// TwinCAT 3 PLC project FsCommon
// Title: FsCommon
// Company: FisoThemes
// Author: Goodwill Mzumala
// ProjectVersion: 0.7.0
// Description: A library that contains common utilites and definitiions to streamline and standardise the development of PLC applications.
// ProgramVersion: 3.1.4023.0
// libraries:
//   SysTarget, * (System)
//   Tc2_Math, * (Beckhoff Automation GmbH)
//   Tc2_Standard, * (Beckhoff Automation GmbH)
//   Tc2_System, * (Beckhoff Automation GmbH)
//   Tc3_Module, * (Beckhoff Automation GmbH)
// project tree:
//   DUTs/ E_Accessor.TcTLEO, E_Comparison.TcTLEO, E_AddressMemoryArea.TcTLEO, E_OperatingSystem.TcTLEO, E_ProcessorArchitecture.TcTLEO, ST_ArrayIterator.TcDUT, T_ArrayIterator.TcDUT, T_Path.TcDUT, T_TypeID.TcDUT, T_WPath.TcDUT, U_Primitive.TcDUT, T_Char.TcDUT, T_MaxWString.TcDUT, T_WChar.TcDUT, T_Generic.TcDUT, T_TaskNameString.TcDUT, T_TypeClass.TcDUT, T_PlcAppSysInfo.TcDUT, T_Position.TcDUT, T_QueryInterface.TcDUT, T_Size.TcDUT, T_VarInfo.TcDUT, U_Pointer.TcDUT
//   DUTs/Primitives/ F32.TcDUT, F64.TcDUT, I16.TcDUT, I32.TcDUT, I64.TcDUT, I8.TcDUT, U16.TcDUT, U32.TcDUT, U64.TcDUT, U8.TcDUT
//   GVLs/ GVL_TypeValueLimits.TcGVL
//   ITFs/ I_ChangeDetector.TcIO, I_PlcTaskInformation.TcIO, I_Destructable.TcIO, I_Runnable.TcIO
//   PARAMs/ PARAM_Constants.TcGVL
//   / PlcTask.TcTTO
//   POUs/Bounds/ F_GetBoolArrayUpperBound.TcPOU, F_GetByteArrayUpperBound.TcPOU, F_GetDateAndTimeArrayUpperBound.TcPOU, F_GetDateArrayUpperBound.TcPOU, F_GetDIntArrayUpperBound.TcPOU, F_GetDWordArrayUpperBound.TcPOU, F_GetIntArrayUpperBound.TcPOU, F_GetInterfaceArrayLowerBound.TcPOU, F_GetInterfaceArrayUpperBound.TcPOU, F_GetLIntArrayUpperBound.TcPOU, F_GetLRealArrayUpperBound.TcPOU, F_GetLTimeArrayUpperBound.TcPOU, F_GetLWordArrayUpperBound.TcPOU, F_GetMaxStringArrayLowerBound.TcPOU, F_GetMaxStringArrayUpperBound.TcPOU, F_GetMaxWStringArrayLowerBound.TcPOU, F_GetMaxWStringArrayUpperBound.TcPOU, F_GetPointerArrayUpperBound.TcPOU, F_GetRealArrayUpperBound.TcPOU, F_GetRunnableArrayLowerBound.TcPOU, F_GetRunnableArrayUpperBound.TcPOU, F_GetSIntArrayUpperBound.TcPOU, F_GetStringArrayUpperBound.TcPOU, F_GetTimeArrayUpperBound.TcPOU, F_GetTimeOfDayArrayUpperBound.TcPOU, F_GetUDIntArrayUpperBound.TcPOU, F_GetUIntArrayUpperBound.TcPOU, F_GetULIntArrayUpperBound.TcPOU, F_GetUSIntArrayUpperBound.TcPOU, F_GetUXIntArrayUpperBound.TcPOU, F_GetWordArrayUpperBound.TcPOU, F_GetWStringArrayLowerBound.TcPOU, F_GetStringArrayLowerBound.TcPOU, F_GetPointerArrayLowerBound.TcPOU, F_GetTimeOfDayArrayLowerBound.TcPOU, F_GetDateAndTimeArrayLowerBound.TcPOU, F_GetDateArrayLowerBound.TcPOU, F_GetTimeArrayLowerBound.TcPOU, F_GetRealArrayLowerBound.TcPOU, F_GetLRealArrayLowerBound.TcPOU, F_GetLTimeArrayLowerBound.TcPOU, F_GetUDIntArrayLowerBound.TcPOU, F_GetULIntArrayLowerBound.TcPOU, F_GetUXIntArrayLowerBound.TcPOU, F_GetUSIntArrayLowerBound.TcPOU, F_GetDIntArrayLowerBound.TcPOU, F_GetLIntArrayLowerBound.TcPOU, F_GetUIntArrayLowerBound.TcPOU, F_GetWStringArrayUpperBound.TcPOU, F_GetXIntArrayLowerBound.TcPOU, F_GetSIntArrayLowerBound.TcPOU, F_GetByteArrayLowerBound.TcPOU, F_GetBoolArrayLowerBound.TcPOU, F_GetLWordArrayLowerBound.TcPOU, F_GetIntArrayLowerBound.TcPOU, F_GetXIntArrayUpperBound.TcPOU, F_GetXWordArrayLowerBound.TcPOU, F_GetWordArrayLowerBound.TcPOU, F_GetDWordArrayLowerBound.TcPOU, F_GetXWordArrayUpperBound.TcPOU
//   POUs/Conversions/ F_DintToSize.TcPOU, F_IntToSize.TcPOU, F_PositionToSize.TcPOU (not stored), F_SizeToDint.TcPOU (not stored), F_SizeToInt.TcPOU (not stored), F_SizeToPosition.TcPOU, F_ULintToPosition.TcPOU
//   POUs/ FB_PlcTaskInformation.TcPOU, FB_RandomNumberGenerator.TcPOU, FB_ValueChangeDetector.TcPOU, FB_PlcTaskCycleChangeDetector.TcPOU, F_AllAreFalse.TcPOU, F_AllocateMemory.TcPOU, F_AnyAreTrue.TcPOU, F_AnyAreFalse.TcPOU, F_AreSameTypeFromInterfaces.TcPOU, F_ExtractPointerFromInterface.TcPOU, F_ExtractVariableNameFromPath.TcPOU, F_GetAddressMemoryArea.TcPOU, F_GetCpuCycleCounter.TcPOU, F_GetCurrentTaskCycleTime.TcPOU, F_GetCurrentPlcTaskInformation.TcPOU, F_GetCurrentTaskIndex.TcPOU, F_GetInf.TcPOU, F_GetMemorySegment.TcPOU, F_GetNaN.TcPOU, F_GetAddressFromInterface.TcPOU, F_DeallocateMemory.TcPOU, F_GetNumberOfPlcTasks.TcPOU, F_GetTypeID.TcPOU, F_GetTypeIDFromGeneric.TcPOU, F_GetVariablePathByAddress.TcPOU, F_GetVariablePath.TcPOU, F_Hash.TcPOU, F_AllAreTrue.TcPOU, F_IsPointerToFunctionBlock.TcPOU, F_IsPointerToInterface.TcPOU, F_IsReadablePointer.TcPOU, F_Lerp.TcPOU, F_ResetOnTrue.TcPOU, F_RunAllRunnables.TcPOU, F_SearchMemory.TcPOU, F_SetDecimalPlaces.TcPOU, F_SetOnFalse.TcPOU, F_SwapMemory.TcPOU, FB_TcComIecApplicationInfo.TcPOU, F_GetTypeNameByAddress.TcPOU, F_GetTypeName.TcPOU, F_GetTypeNameByPath.TcPOU, F_TcComIecApplicationInfo.TcPOU, F_RoundToDecimalPlaces.TcPOU, F_TruncateNumber.TcPOU, F_TryDerefPointer.TcPOU, P_GetSystemInformation.TcPOU, PLAYGROUND.TcPOU
//   Project Information/ F_GetCompany.TcPOU, F_GetTitle.TcPOU, F_GetVersion.TcPOU
//   Version/ Global_Version.TcGVL
// real-time tasks:
//   TASK PlcTask: cycle T#10ms, priority 20, ADS port 350
//   TASK PlcTestTask: cycle T#10ms, priority 21, ADS port 351

CONFIGURATION FsCommon
    RESOURCE PLC ON TwinCAT3
        TASK PlcTask(INTERVAL := T#10ms, PRIORITY := 20);
        PROGRAM PLAYGROUND WITH PlcTask : PLAYGROUND;
    END_RESOURCE
END_CONFIGURATION

// ---- DUTs/E_Accessor.TcTLEO
// An enum that can be used to represent getters and setters.
{attribute 'qualified_only'}
{attribute 'to_string'}
TYPE E_Accessor :
(
	_ := 0, // Unknown/Invalid
	Get,
	Set
)BYTE;
END_TYPE

// ---- DUTs/E_Comparison.TcTLEO
// Comparison enum.
{attribute 'qualified_only'}
{attribute 'to_string'}
TYPE E_Comparison :
(
	_ := 0, // Unknown/Invalid
	Less,
	Equal,
	Greater
)BYTE;
END_TYPE

// ---- DUTs/E_AddressMemoryArea.TcTLEO
// An enum to specify the memory area type of an address.
{attribute 'qualified_only'}
{attribute 'to_string'}
TYPE E_AddressMemoryArea :
(
	_ 		:= 0, 	// Unknown/Invalid.
	Static	:= 1, 	// Static memory.
	Dynamic	:= 2, 	// Dynamic memory.
	CNC		:= 3	// CNC static memory.
)BYTE;
END_TYPE

// ---- DUTs/E_OperatingSystem.TcTLEO
// Operating system used by the machine.
{attribute 'qualified_only'}
{attribute 'to_string'}
TYPE E_OperatingSystem :
(
	_ 			:= 0, 		// Invalid/Unknown/Ininitialised
	Windows,				// Windows OS
	Linux		:= 5,		// Linux
	VxWorks,				// VxWorks RTOS
	QNX,					// Blackberry QNX Embedded OS
	uCOS					// Micro-Controller Operating Systems by Jean J. Labrosse (1991)
) BYTE;
END_TYPE

// ---- DUTs/E_ProcessorArchitecture.TcTLEO
// Processor used by the machine.
{attribute 'qualified_only'}
{attribute 'to_string'}
TYPE E_ProcessorArchitecture :
(
	_ 			:= 0, 	// Invalid/Unknown/Ininitialised
	X86,				// X86 Processor
	ARM,				// ARM Processor
	PowerPC,			// PowerPC Processor
	MIPS				// MIPS processor (as of March 2021 MIPS Technology has moved to RISC-V)
)BYTE;
END_TYPE

// ---- DUTs/ST_ArrayIterator.TcDUT
// Struct for iterating over an array, encapsulating the starting and ending indices.
TYPE ST_ArrayIterator :
STRUCT
    Index   : T_Position := 0; // The current index for the loop, initialised to 0.
    End     : T_Position := -1; // The ending index for the loop, initialised to -1 indicating uninitialised.
END_STRUCT
END_TYPE

// ---- DUTs/T_ArrayIterator.TcDUT
// Type alias for an array iterator.
TYPE T_ArrayIterator : ST_ArrayIterator; END_TYPE

// ---- DUTs/T_Path.TcDUT
// Type alias for a file path string.
// [note] Change the maximum length of the path string in `PARAM_Constants.PATH_LENGTH`
TYPE T_Path : STRING(PARAM_Constants.PATH_LENGTH); END_TYPE

// ---- DUTs/T_TypeID.TcDUT
TYPE T_TypeID : __UXINT; END_TYPE

// ---- DUTs/T_WPath.TcDUT
// Type alias for a file path wide string.
// [note] Change the maximum length of the path string in `PARAM_Constants.PATH_LENGTH`
TYPE T_WPath : WSTRING(PARAM_Constants.PATH_LENGTH); END_TYPE

// ---- DUTs/U_Primitive.TcDUT
// U_Primitive is a union type that can represent various primitive data types.
// This type is useful for handling different kinds of data in a unified manner,
// allowing easy access and manipulation of basic data types and pointers.
TYPE U_Primitive :
UNION
    bBool           : BOOL;                  // Boolean value.
    nByte           : BYTE;                  // 8-bit unsigned integer.
    nWord           : WORD;                  // 16-bit unsigned integer.
    nDWord          : DWORD;                 // 32-bit unsigned integer.
    nLWord          : LWORD;                 // 64-bit unsigned integer.
    nXWord          : __XWORD;               // CPU register size integer (platform-dependent).
    nSInt           : SINT;                  // 8-bit signed integer.
    nInt            : INT;                   // 16-bit signed integer.
    nDInt           : DINT;                  // 32-bit signed integer.
    nLInt           : LINT;                  // 64-bit signed integer.
    nXInt           : __XINT;                // CPU register size signed integer (platform-dependent).
    nUSInt          : USINT;                 // 8-bit unsigned integer.
    nUInt           : UINT;                  // 16-bit unsigned integer.
    nUDInt          : UDINT;                 // 32-bit unsigned integer.
    nULInt          : ULINT;                 // 64-bit unsigned integer.
    nUXInt          : __UXINT;               // CPU register size unsigned integer (platform-dependent).
    fReal           : REAL;                  // 32-bit floating point.
    fLReal          : LREAL;                 // 64-bit floating point.
    tTime           : TIME;                  // Duration in milliseconds.
    tLTime          : LTIME;                 // Duration in nanoseconds.
    dDate           : DATE;                  // Date.
    dtDateAndTime   : DATE_AND_TIME;         // Combined date and time.
    todTimeOfDay    : TIME_OF_DAY;           // Time of day.
    ipInterface     : __SYSTEM.IQueryInterface; // Interface pointer.
    uPointer        : U_Pointer;             // Various pointer types.
    pVoidPointer    : PVOID;                 // Generic pointer to any type.
    arBytes         : ARRAY[0..7] OF BYTE;   // Array of bytes (8 bytes).
END_UNION
END_TYPE

// ---- DUTs/T_Char.TcDUT
// Type alias for a single character string.
TYPE T_Char : STRING(1); END_TYPE

// ---- DUTs/T_MaxWString.TcDUT
// Type alias for a wide string with a maximum length of 255 characters.
TYPE T_MaxWString : WSTRING(255); END_TYPE

// ---- DUTs/T_WChar.TcDUT
// Type alias for a single wide character string.
TYPE T_WChar : WSTRING(1); END_TYPE

// ---- DUTs/T_Generic.TcDUT
// Type alias for a generic type, __SYSTEM.AnyType.
TYPE T_Generic : __SYSTEM.AnyType; END_TYPE

// ---- DUTs/T_TaskNameString.TcDUT
TYPE T_TaskNameString : STRING(63); END_TYPE

// ---- DUTs/T_TypeClass.TcDUT
TYPE T_TypeClass : __SYSTEM.TYPE_CLASS; END_TYPE

// ---- DUTs/Primitives/F32.TcDUT
TYPE F32 : REAL; END_TYPE

// ---- DUTs/Primitives/F64.TcDUT
TYPE F64 : LREAL; END_TYPE

// ---- DUTs/Primitives/I16.TcDUT
TYPE I16 : INT; END_TYPE

// ---- DUTs/Primitives/I32.TcDUT
TYPE I32 : DINT; END_TYPE

// ---- DUTs/Primitives/I64.TcDUT
TYPE I64 : LINT; END_TYPE

// ---- DUTs/Primitives/I8.TcDUT
TYPE I8 : SINT; END_TYPE

// ---- DUTs/Primitives/U16.TcDUT
TYPE U16 : UINT; END_TYPE

// ---- DUTs/Primitives/U32.TcDUT
TYPE U32 : UDINT; END_TYPE

// ---- DUTs/Primitives/U64.TcDUT
TYPE U64 : ULINT; END_TYPE

// ---- DUTs/Primitives/U8.TcDUT
TYPE U8 : BYTE; END_TYPE

// ---- DUTs/T_PlcAppSysInfo.TcDUT
// Type alias for a struct PLC application system information.
TYPE T_PlcAppSysInfo : PlcAppSystemInfo; END_TYPE

// ---- DUTs/T_Position.TcDUT
// Type alias for represeting position.
TYPE T_Position : LINT; END_TYPE

// ---- DUTs/T_QueryInterface.TcDUT
TYPE T_QueryInterface : __SYSTEM.IQueryInterface; END_TYPE

// ---- DUTs/T_Size.TcDUT
// Type alias for represeting size or capacity.
TYPE T_Size : UDINT; END_TYPE

// ---- DUTs/T_VarInfo.TcDUT
// Alias for __SYSTEM.VAR_INFO.
// [use] Stores variable information.
TYPE T_VarInfo : __SYSTEM.VAR_INFO; END_TYPE

// ---- DUTs/U_Pointer.TcDUT
// U_Pointer is a union type that can represent various pointer types.
// This type is useful for handling different kinds of pointers in a unified manner,
// allowing easy access and manipulation of different data types through pointers.
TYPE U_Pointer :
UNION
    pBool           : POINTER TO BOOL;                 // Pointer to a Boolean value.
    pByte           : POINTER TO BYTE;                 // Pointer to an 8-bit unsigned integer.
    pWord           : POINTER TO WORD;                 // Pointer to a 16-bit unsigned integer.
    pDWord          : POINTER TO DWORD;                // Pointer to a 32-bit unsigned integer.
    pLWord          : POINTER TO LWORD;                // Pointer to a 64-bit unsigned integer.
    pXWord          : POINTER TO __XWORD;              // Pointer to a CPU register size integer (platform-dependent).
    pSInt           : POINTER TO SINT;                 // Pointer to an 8-bit signed integer.
    pInt            : POINTER TO INT;                  // Pointer to a 16-bit signed integer.
    pDInt           : POINTER TO DINT;                 // Pointer to a 32-bit signed integer.
    pLInt           : POINTER TO LINT;                 // Pointer to a 64-bit signed integer.
    pXInt           : POINTER TO __XINT;               // Pointer to a CPU register size signed integer (platform-dependent).
    pUSInt          : POINTER TO USINT;                // Pointer to an 8-bit unsigned integer.
    pUInt           : POINTER TO UINT;                 // Pointer to a 16-bit unsigned integer.
    pUDInt          : POINTER TO UDINT;                // Pointer to a 32-bit unsigned integer.
    pULInt          : POINTER TO ULINT;                // Pointer to a 64-bit unsigned integer.
    pUXInt          : POINTER TO __UXINT;              // Pointer to a CPU register size unsigned integer (platform-dependent).
    pReal           : POINTER TO REAL;                 // Pointer to a 32-bit floating point.
    pLReal          : POINTER TO LREAL;                // Pointer to a 64-bit floating point.
    pString         : POINTER TO STRING;               // Pointer to a string.
    pMaxString      : POINTER TO Tc2_System.T_MaxString; // Pointer to a max length string.
    pWString        : POINTER TO WSTRING;              // Pointer to a wide string.
    pMaxWString     : POINTER TO T_MaxWString;         // Pointer to a max length wide string.
    pTime           : POINTER TO TIME;                 // Pointer to a duration in milliseconds.
    pLTime          : POINTER TO LTIME;                // Pointer to a duration in nanoseconds.
    pDate           : POINTER TO DATE;                 // Pointer to a date.
    pDateAndTime    : POINTER TO DATE_AND_TIME;        // Pointer to a combined date and time.
    pTimeOfDay      : POINTER TO TIME_OF_DAY;          // Pointer to a time of day.
    pInterface      : POINTER TO __SYSTEM.IQueryInterface; // Pointer to an interface.
    pNested         : POINTER TO U_Pointer;            // Pointer to another U_Pointer.
    pVoid           : PVOID;                           // Generic pointer to any type.
    nSignedInteger  : __XINT;                          // CPU register size signed integer.
    nUnsignedInteger: __UXINT;                         // CPU register size unsigned integer.
    nWord           : __XWORD;                         // CPU register size integer (platform-dependent).
END_UNION
END_TYPE

// ---- GVLs/GVL_TypeValueLimits.TcGVL
{attribute 'qualified_only'}
VAR_GLOBAL CONSTANT
    // Minimum and maximum values for BYTE type
    BYTE_MIN        : BYTE           := 0;          // Minimum value for BYTE
    BYTE_MAX        : BYTE           := 255;        // Maximum value for BYTE
    
    // Minimum and maximum values for WORD type
    WORD_MIN        : WORD           := 16#0;       // Minimum value for WORD
    WORD_MAX        : WORD           := 16#FFFF;    // Maximum value for WORD
    
    // Minimum and maximum values for DWORD type
    DWORD_MIN       : DWORD          := 16#0;       // Minimum value for DWORD
    DWORD_MAX       : DWORD          := 16#FFFFFFFF;// Maximum value for DWORD
    
    // Minimum and maximum values for LWORD type
    LWORD_MIN       : LWORD          := 16#0;				 // Minimum value for LWORD
    LWORD_MAX       : LWORD          := 16#FFFFFFFFFFFFFFFF; // Maximum value for LWORD
    
    // Minimum and maximum values for SINT type
    SINT_MIN        : SINT           := -128;       // Minimum value for SINT
    SINT_MAX        : SINT           := +127;       // Maximum value for SINT
    
    // Minimum and maximum values for UINT type
    UINT_MIN        : UINT           := 0;          // Minimum value for UINT
    UINT_MAX        : UINT           := 65535;      // Maximum value for UINT
    
    // Minimum and maximum values for INT type
    INT_MIN         : INT            := -32768;     // Minimum value for INT
    INT_MAX         : INT            := +32767;     // Maximum value for INT
    
    // Minimum and maximum values for UDINT type
    UDINT_MIN       : UDINT          := 0;				// Minimum value for UDINT
    UDINT_MAX       : UDINT          := 4_294_967_295; 	// Maximum value for UDINT
    
    // Minimum and maximum values for DINT type
    DINT_MIN        : DINT           := -2_147_483_648; // Minimum value for DINT
    DINT_MAX        : DINT           := +2_147_483_647; // Maximum value for DINT
    
    // Minimum and maximum values for ULINT type
    ULINT_MIN       : ULINT          := 0;							// Minimum value for ULINT
    ULINT_MAX       : ULINT          := 18_446_744_073_709_551_615; // Maximum value for ULINT
    
    // Minimum and maximum values for LINT type
    LINT_MIN        : LINT           := -9_223_372_036_854_775_808; // Minimum value for LINT
    LINT_MAX        : LINT           := +9_223_372_036_854_775_807; // Maximum value for LINT
    
    // Minimum and maximum values for REAL type
    REAL_MIN        : REAL           := -3.402823E+38; // Minimum value for REAL
    REAL_MAX        : REAL           := +3.402823E+38; // Maximum value for REAL
    
    // Minimum and maximum values for LREAL type
    LREAL_MIN       : LREAL          := -1.7976931348623158E+308; // Minimum value for LREAL
    LREAL_MAX       : LREAL          := +1.7976931348623158E+308; // Maximum value for LREAL
    
    // Minimum and maximum values for TIME type
    TIME_MIN        : TIME           := T#0S;       // Minimum value for TIME
    TIME_MAX        : TIME           := T#49D17H2M47S295MS; // Maximum value for TIME
    
    // Minimum and maximum values for LTIME type
    LTIME_MIN       : LTIME          := LTIME#0S;   // Minimum value for LTIME
    LTIME_MAX       : LTIME          := LTIME#213503D23H34M33S709MS551US615NS; // Maximum value for LTIME
    
    // Minimum and maximum values for DATE type
    DATE_MIN        : DATE           := D#1970-01-01; // Minimum value for DATE
    DATE_MAX        : DATE           := D#2106-02-07; // Maximum value for DATE
    
    // Minimum and maximum values for DT (DateTime) type
    DT_MIN          : DT             := DT#1970-1-1-0:0:0; // Minimum value for DT
    DT_MAX          : DT             := DT#2106-02-07-06:28:15; // Maximum value for DT
    
    // Minimum and maximum values for TOD (Time of Day) type
    TOD_MIN         : TOD            := TOD#0:0:0; // Minimum value for TOD
    TOD_MAX         : TOD            := TOD#23:59:59.999; // Maximum value for TOD
    
    // Minimum and maximum values for T_Size type
    T_SIZE_MIN      : T_Size         := UDINT_MIN;  // Minimum value for T_Size
    T_SIZE_MAX      : T_Size         := UDINT_MAX;  // Maximum value for T_Size
    
    // Minimum and maximum values for T_Position type
    T_POSITION_MIN  : T_Position     := LINT_MIN;   // Minimum value for T_Position
    T_POSITION_MAX  : T_Position     := LINT_MAX;   // Maximum value for T_Position
END_VAR

// ---- PARAMs/PARAM_Constants.TcGVL
// Main parameters for the library.
{attribute 'qualified_only'}
VAR_GLOBAL CONSTANT
	PATH_LENGTH			: __UXINT := 300; // String length of path type.
END_VAR

// ---- Version/Global_Version.TcGVL
{attribute 'TcGenerated'}
{attribute 'no-analysis'}
{attribute 'linkalways'}
// This function has been automatically generated from the project information.
VAR_GLOBAL CONSTANT
	{attribute 'const_non_replaced'}
	stLibVersion_FsCommon : ST_LibVersion := (iMajor := 0, iMinor := 7, iBuild := 0, iRevision := 0, nFlags := 0, sVersion := '0.7.0');
END_VAR

// ---- ITFs/I_ChangeDetector.TcIO
// Interface for indicating that an object is for detecting the change of some object/value.
INTERFACE I_ChangeDetector EXTENDS __SYSTEM.IQueryInterface

// Indicates if the object has changed.
// [get] Returns flag indicating of object has changed.
PROPERTY HasChanged : BOOL
GET
END_GET
END_PROPERTY

END_INTERFACE

// ---- ITFs/I_PlcTaskInformation.TcIO
// Interface for accessing information about a PLC task.
INTERFACE I_PlcTaskInformation EXTENDS __SYSTEM.IQueryInterface

// Task's ADS Port.
// [get] Returns the referenced task's ADS port.
PROPERTY AdsPort : UINT
GET
END_GET
END_PROPERTY

// The task's cycle counter.
// [note] This refers to the actual system task and not to the task reference of the PLC project.
// [get] Returns the task's cycle counter.
PROPERTY CycleCount : UDINT
GET
END_GET
END_PROPERTY

// The cycle time of the task.
// [get] Returns the cycle time.
PROPERTY CycleTime : LTIME
GET
END_GET
END_PROPERTY

// Indicates whether the cycle time has been exceeded.
// [get] Returns TRUE if the cycle time has been exceeded.
PROPERTY CycleTimeExceeded : BOOL
GET
END_GET
END_PROPERTY

// Indicates if the origin of the current call is declared with the attribute 'TcCallAfterOutputUpdate'.
// [get] Returns TRUE if current call is declared with the attribute 'TcCallAfterOutputUpdate'.
PROPERTY HasCallAfterOutputUpdateAttribute : BOOL
GET
END_GET
END_PROPERTY

// The index of the task.
// [get] Returns the index.
PROPERTY Index : DINT
GET
END_GET
END_PROPERTY

// Indicates if it is the first cycle of the task.
// [get] Returns TRUE if it is the first cycle.
PROPERTY IsFirstCycle : BOOL
GET
END_GET
END_PROPERTY

// Time the previous cycle took to complete execution.
// [get] Returns the last exection time.
PROPERTY LastCycleExecutionTime : LTIME
GET
END_GET
END_PROPERTY

// The name of the task.
// [get] Returns the task name.
PROPERTY Name : T_TaskNameString
GET
END_GET
END_PROPERTY

// The object ID of the task reference, from which the PLC program is called.
// [get] Returns the object ID.
PROPERTY ObjectId : OTCID
GET
END_GET
END_PROPERTY

// The priority of the task.
// [get] Returns the priority.
PROPERTY Priority : UINT
GET
END_GET
END_PROPERTY

// Indicates whether the real-time time limit has been exceeded on a mixed core (Windows + real-time on one core).
// [get] Returns true if the real-time time limit has been exceeded.
PROPERTY RTTimeLimitExceeded : BOOL
GET
END_GET
END_PROPERTY

END_INTERFACE

// ---- ITFs/I_Destructable.TcIO
// Interface to indicate that an object has resources that need to be released.
INTERFACE I_Destructable EXTENDS __SYSTEM.IQueryInterface

METHOD FB_exit : BOOL
VAR_INPUT
	bInCopyCode : BOOL; // if TRUE, the exit method is called for exiting an instance that is copied afterwards (online change).
END_VAR
END_METHOD

END_INTERFACE

// ---- ITFs/I_Runnable.TcIO
(*
Interface for objects that expose a cyclic :meth:`Run` method.

Use :func:`F_IsRunnable` to check whether an object implements this interface
at runtime before calling :meth:`Run`.
*)
INTERFACE I_Runnable EXTENDS __SYSTEM.IQueryInterface

(* Executes one cycle of the object's logic. Call only once per cycle on a single task. *)
METHOD Run
VAR_INPUT
END_VAR
END_METHOD

END_INTERFACE

// ---- POUs/PLAYGROUND.TcPOU
{attribute 'no_explicit_call' := 'direct call for this program is not allowed'} 
PROGRAM INTERNAL PLAYGROUND
VAR
	sTypeName,
	Str1, Str2				: T_MaxString;
	pFound 					: POINTER TO STRING;
	uPointer 				: U_Pointer := (pString := ADR(Str1));
	bStart 					: BOOL := TRUE;
	nCpuCycle				: ULINT;
	eOpSys 					: E_OperatingSystem;
	eProcArc				: E_ProcessorArchitecture;
	ipTaskInfo 				: I_PlcTaskInformation;
	fbTaskInfo 				: FB_PlcTaskInformation;
	fbTaskCycleChanged		: FB_PlcTaskCycleChangeDetector(0); 
	nHash 					: DWORD;
	AmsPort 				: Tc2_System.T_AmsPort;
	CycleTime, LastExecTime : LTIME;
	i, j, Count, Size 		: T_Size;
	Str 					: STRING := '123456789';
	fbGenRand				: FB_RandomNumberGenerator(0);
	nRand1, nRand2			: LINT;
	fRand1, fRand2			: LREAL;
END_VAR

sTypeName := F_GetTypeName(pFound);
nHash := F_Hash(ADR(Str), F_PositionToSize(LEN(Str)), 0);
nCpuCycle		:= F_GetCpuCycleCounter();
eProcArc 		:= P_GetSystemInformation.ProcessorArchitecture;
eOpSys 			:= P_GetSystemInformation.OperatingSystem;
AmsPort 		:= F_GetCurrentPlcTaskInformation().AdsPort;
CycleTime 		:= F_GetCurrentPlcTaskInformation().CycleTime;
LastExecTime 	:= F_GetCurrentPlcTaskInformation().LastCycleExecutionTime;
Count 			:= F_GetCurrentPlcTaskInformation().CycleCount;
Size 			:= F_GetNumberOfPlcTasks();

nRand1 := fbGenRand.NextInt();
nRand2 := fbGenRand.NextRangedInt(10, -10);
fRand1 := fbGenRand.NextReal();
fRand2 := F_SetDecimalPlaces(fbGenRand.NextRangedReal(-5.8, 9.432), 2);

pFound := F_SearchMemory(ADR(Str1), F_IntToSize(LEN(Str1)), ADR(Str2), F_IntToSize(LEN(Str2)));

IF NOT F_ResetOnTrue(bStart) THEN RETURN; END_IF

i := SEL(fbTaskCycleChanged.HasChanged, i, i + 1);
j := SEL(fbTaskCycleChanged.HasChanged, j, j + 1);

END_PROGRAM

// ---- POUs/FB_PlcTaskInformation.TcPOU
// Retrieves PLC Task information.
// [note] if not explicitly defined, the default task index is the task the function block is instatiated on. 
{attribute 'enable_dynamic_creation'}
{attribute 'no_explicit_call' := 'direct call for this function block is not allowed'}
FUNCTION_BLOCK FINAL FB_PlcTaskInformation IMPLEMENTS I_PlcTaskInformation
VAR
	_nTaskIndex : DINT;
END_VAR

// Task's ADS Port.
// [get] Returns the referenced task's ADS port.
PROPERTY AdsPort : Tc2_System.T_AmsPort
GET
AdsPort := TwinCAT_SystemInfoVarList._TaskInfo[THIS^._nTaskIndex].AdsPort;
END_GET
END_PROPERTY

// The task's cycle counter.
// [note] This refers to the actual system task and not to the task reference of the PLC project.
// [get] Returns the task's cycle counter.
PROPERTY CycleCount : UDINT
GET
CycleCount := TwinCAT_SystemInfoVarList._TaskInfo[THIS^._nTaskIndex].CycleCount;
END_GET
END_PROPERTY

// The cycle time of the task.
// [get] Returns the cycle time.
PROPERTY CycleTime : LTIME
GET
CycleTime := TO_LTIME(TwinCAT_SystemInfoVarList._TaskInfo[THIS^._nTaskIndex].CycleTime * 100);
END_GET
END_PROPERTY

// Indicates whether the cycle time has been exceeded.
// [get] Returns TRUE if the cycle time has been exceeded.
PROPERTY CycleTimeExceeded : BOOL
GET
CycleTimeExceeded := TwinCAT_SystemInfoVarList._TaskInfo[THIS^._nTaskIndex].CycleTimeExceeded;
END_GET
END_PROPERTY

{attribute 'hide'}
METHOD FB_init : BOOL
VAR_INPUT
	bInitRetains : BOOL; // if TRUE, the retain variables are initialized (warm start / cold start)
	bInCopyCode : BOOL;  // if TRUE, the instance afterwards gets moved into the copy code (online change)
END_VAR
VAR
	fbGetCurrentTaskIndex : Tc2_System.GETCURTASKINDEX;
END_VAR
// Return if online change.
IF bInCopyCode THEN RETURN; END_IF

fbGetCurrentTaskIndex(Index => THIS^._nTaskIndex);
END_METHOD

// Indicates if the origin of the current call is declared with the attribute 'TcCallAfterOutputUpdate'.
// [get] Returns TRUE if current call is declared with the attribute 'TcCallAfterOutputUpdate'.
PROPERTY HasCallAfterOutputUpdateAttribute : BOOL
GET
HasCallAfterOutputUpdateAttribute := TwinCAT_SystemInfoVarList._TaskInfo[THIS^._nTaskIndex].InCallAfterOutputUpdate;
END_GET
END_PROPERTY

// The index of the task.
// [get] Returns the index.
// [set] The index of the task to retrieve information from.
PROPERTY Index : DINT
GET
Index := THIS^._nTaskIndex;
END_GET
SET
THIS^._nTaskIndex := LIMIT(1, Index, F_SizeToDint(F_GetNumberOfPlcTasks()));
END_SET
END_PROPERTY

// Indicates if it is the first cycle of the task.
// [get] Returns TRUE if it is the first cycle.
PROPERTY IsFirstCycle : BOOL
GET
IsFirstCycle := TwinCAT_SystemInfoVarList._TaskInfo[THIS^._nTaskIndex].FirstCycle;
END_GET
END_PROPERTY

// Time the previous cycle took to complete execution.
// [get] Returns the last exection time.
PROPERTY LastCycleExecutionTime : LTIME
GET
LastCycleExecutionTime := TO_LTIME(TwinCAT_SystemInfoVarList._TaskInfo[THIS^._nTaskIndex].LastExecTime * 100);
END_GET
END_PROPERTY

// The name of the task.
// [get] Returns the task name.
PROPERTY Name : T_TaskNameString
GET
Name := TwinCAT_SystemInfoVarList._TaskInfo[THIS^._nTaskIndex].TaskName;
END_GET
END_PROPERTY

// The object ID of the task reference, from which the PLC program is called.
// [get] Returns the object ID.
PROPERTY ObjectId : OTCID
GET
ObjectId := TwinCAT_SystemInfoVarList._TaskInfo[THIS^._nTaskIndex].ObjId;
END_GET
END_PROPERTY

// The priority of the task.
// [get] Returns the priority.
PROPERTY Priority : UINT
GET
Priority := TwinCAT_SystemInfoVarList._TaskInfo[THIS^._nTaskIndex].Priority;
END_GET
END_PROPERTY

// Indicates whether the real-time time limit has been exceeded on a mixed core (Windows + real-time on one core).
// [get] Returns true if the real-time time limit has been exceeded.
PROPERTY RTTimeLimitExceeded : BOOL
GET
RTTimeLimitExceeded := TwinCAT_SystemInfoVarList._TaskInfo[THIS^._nTaskIndex].RTViolation;
END_GET
END_PROPERTY

END_FUNCTION_BLOCK

// ---- POUs/F_GetNumberOfPlcTasks.TcPOU
// Retrieves the number of PLC tasks available in the system.
FUNCTION F_GetNumberOfPlcTasks : T_Size // The number of PLC tasks.

F_GetNumberOfPlcTasks := SIZEOF(TwinCAT_SystemInfoVarList._TaskInfo) / SIZEOF(PlcTaskSystemInfo);

END_FUNCTION

// ---- POUs/FB_PlcTaskCycleChangeDetector.TcPOU
// Detects if the current PLC task cycle has changed.
// If index of the initialiser less than 1, the task index the object is instatiated on is watched.
// [init] <Instance Name> : FB_PlcTaskCycleChangeDetector(<Task Index>);
{attribute 'enable_dynamic_creation'}
{attribute 'no_explicit_call' := 'direct call for this function block is not allowed'}
FUNCTION_BLOCK FINAL FB_PlcTaskCycleChangeDetector IMPLEMENTS I_ChangeDetector
VAR
	_nTaskIndex 		: DINT	:= 1;
	_nLastCycleChecked 	: UDINT := GVL_TypeValueLimits.UDINT_MAX; // The last cycle checked for change-in-plc-cycle.
END_VAR

// The task's current cycle counter.
// [note] This refers to the actual system task and not to the task reference of the PLC project.
// [get] Returns the current task's cycle counter.
PROPERTY CurrentCycle : UDINT
GET
CurrentCycle := TwinCAT_SystemInfoVarList._TaskInfo[THIS^._nTaskIndex].CycleCount;
END_GET
END_PROPERTY

{attribute 'hide'}
METHOD FB_init : BOOL
VAR_INPUT
	bInitRetains 	: BOOL; // if TRUE, the retain variables are initialized (warm start / cold start)
	bInCopyCode 	: BOOL; // if TRUE, the instance afterwards gets moved into the copy code (online change)
	nTaskIndex 		: DINT; // Index of task to monitor. 0 or less = Task the object is instatiated at.
END_VAR
// Return if online change.
IF bInCopyCode THEN RETURN; END_IF

THIS^._nTaskIndex := SEL(nTaskIndex > 0,
						 F_GetCurrentPlcTaskInformation().Index,
						 LIMIT(1, nTaskIndex, F_SizeToDint(F_GetNumberOfPlcTasks())));
END_METHOD

// Indicates if the value has changed.
// [get] Returns flag indicating of value has changed.
PROPERTY HasChanged : BOOL
GET
HasChanged := THIS^.CurrentCycle <> THIS^._nLastCycleChecked;
THIS^._nLastCycleChecked := THIS^.CurrentCycle;
END_GET
END_PROPERTY

// Indicates if it is the first cycle of the task.
// [get] Returns TRUE if it is the first cycle.
PROPERTY IsFirstCycle : BOOL
GET
 IsFirstCycle := TwinCAT_SystemInfoVarList._TaskInfo[THIS^._nTaskIndex].FirstCycle;
END_GET
END_PROPERTY

// The last cycle checked for change-in-plc-cycle.
// [get] Returns the last cycle checked.
PROPERTY LastCycleChecked : UDINT
GET
LastCycleChecked := THIS^._nLastCycleChecked;
END_GET
END_PROPERTY

// The index of the task being monitored.
// [get] Returns the index.
// [set] The index of the task to monitor (clamp to a minimum of 1).
PROPERTY TaskIndex : DINT
GET
TaskIndex := THIS^._nTaskIndex;
END_GET
SET
THIS^._nTaskIndex := LIMIT(1, TaskIndex, F_SizeToDint(F_GetNumberOfPlcTasks()));
END_SET
END_PROPERTY

END_FUNCTION_BLOCK

// ---- POUs/F_GetCurrentPlcTaskInformation.TcPOU
// Retrieves the information about the current PLC task.
FUNCTION F_GetCurrentPlcTaskInformation : I_PlcTaskInformation // An instance of I_PlcTaskInformation containing details of the current PLC task.
VAR_STAT
	fbGetCurrentTaskIndex : Tc2_System.GETCURTASKINDEX;
	fbPlcTaskInformation : FB_PlcTaskInformation;
END_VAR

fbGetCurrentTaskIndex();
fbPlcTaskInformation.Index 		:= fbGetCurrentTaskIndex.Index;
F_GetCurrentPlcTaskInformation 	:= fbPlcTaskInformation;

END_FUNCTION

// ---- POUs/FB_RandomNumberGenerator.TcPOU
// Generates pseudo-random numbers.
// [init] <Instance Name> : FB_RandomNumberGenerator(<Initial Seed>);
// [note] The methods in this function block can be called using ADS-RPC.
{attribute 'enable_dynamic_creation'}
{attribute 'no_explicit_call' := 'direct call for this function block is not allowed'}
FUNCTION_BLOCK FINAL FB_RandomNumberGenerator IMPLEMENTS __SYSTEM.IQueryInterface
VAR
	_nSeed : LINT;
END_VAR
VAR_STAT CONSTANT
	_nLGC_M : LINT := LINT#9223372036854775783;
END_VAR

{attribute 'hide'}
METHOD FB_init : BOOL
VAR_INPUT
	bInitRetains 	: BOOL; // if TRUE, the retain variables are initialized (warm start / cold start)
	bInCopyCode 	: BOOL; // if TRUE, the instance afterwards gets moved into the copy code (online change)
	nSeed 			: LINT; // Initial seed value for the generator.
END_VAR
// Return if online change.
IF bInCopyCode THEN RETURN; END_IF

THIS^._nSeed := nSeed;
END_METHOD

// Generates additional entropy based on system timestamp, task time and CPU cycle.
METHOD PRIVATE GetSystemEntropy : LINT // System entropy.
VAR_INPUT
	nSeed : LINT;
END_VAR
GetSystemEntropy := TO_LINT(TO_ULINT(nSeed) XOR Tc2_System.F_GetSystemTime() XOR Tc2_System.F_GetTaskTime() XOR F_GetCpuCycleCounter());
END_METHOD

// LCG formula for updating the seed.
METHOD PRIVATE LinearCongruentialGenerator : LINT // New seed value.
VAR_INPUT
	nSeed : LINT;
END_VAR
LinearCongruentialGenerator := (LINT#6364136223846793005 * nSeed * LINT#1442695040888963407) MOD THIS^._nLGC_M;
END_METHOD

// Generates the next pseudo-random integer.
{attribute 'TcRpcEnable'}
METHOD NextInt : LINT // The next pseudo-random integer.
VAR_INPUT
END_VAR
NextInt := THIS^._nSeed := THIS^.LinearCongruentialGenerator(TO_LINT(TO_ULINT(THIS^._nSeed) XOR TO_ULINT(THIS^.GetSystemEntropy(THIS^._nSeed))));
END_METHOD

// Generates the next pseudo-random integer within the specified range [minimum, maximum].
{attribute 'TcRpcEnable'}
METHOD NextRangedInt : LINT // The next pseudo-random integer within the range.
VAR_INPUT
	nMinimum : LINT; // Minimum value of the range. 
	nMaximum : LINT; // Maximum value of the range.
END_VAR
NextRangedInt := MIN(nMinimum, nMaximum) + (ABS(THIS^.NextInt()) MOD (MAX(nMinimum, nMaximum) - MIN(nMinimum, nMaximum) + 1));
END_METHOD

// Generates the next pseudo-random real number within the specified range [minimum, maximum].
{attribute 'TcRpcEnable'}
METHOD NextRangedReal : LREAL // The next pseudo-random real number within the range.
VAR_INPUT
	fMinimum : LREAL; // Minimum value of the range. 
	fMaximum : LREAL; // Maximum value of the range.
END_VAR
NextRangedReal := MIN(fMinimum, fMaximum) + (ABS(THIS^.NextReal()) * (MAX(fMinimum, fMaximum) - MIN(fMinimum, fMaximum)));
END_METHOD

// Generates the next pseudo-random real number.
{attribute 'TcRpcEnable'}
METHOD NextReal : LREAL // The next pseudo-random real number.
VAR_INPUT
END_VAR
NextReal := TO_LREAL(THIS^.NextInt()) / TO_LREAL(THIS^._nLGC_M + 1);
END_METHOD

END_FUNCTION_BLOCK

// ---- POUs/F_GetCpuCycleCounter.TcPOU
// Gets the CPU's cycle count.
// The value us refreshed every 100ns.
FUNCTION F_GetCpuCycleCounter : ULINT // The current CPU count with in the 100ns refresh rate.
VAR_STAT
	fbGetCpuCounter : Tc2_System.GETCPUCOUNTER;
END_VAR

fbGetCpuCounter();
F_GetCpuCycleCounter := SHL(TO_ULINT(fbGetCpuCounter.cpuCntHiDW), 32) OR fbGetCpuCounter.cpuCntLoDW;

END_FUNCTION

// ---- POUs/F_GetTypeName.TcPOU
// Retrieves the datatype of a given variable as a string.
// [note] Variables allocated in dynamic memory are not supported.
{warning disable C0394}
FUNCTION F_GetTypeName : STRING // The datatype name of the variable as a string.
VAR_INPUT
    Variable : ANY; // The variable whose datatype is to be determined.
END_VAR
VAR_STAT
	nTmp : UDINT := SIZEOF(F_GetTypeName);
END_VAR
VAR
	ipInterface : ITcIecApplicationInfo;
END_VAR

CASE Tc2_System.F_CheckMemoryArea(Variable.pValue, 1) OF
	Tc2_System.E_TcMemoryArea.Dynamic: F_GetTypeName := '<dynamic>';
	Tc2_System.E_TcMemoryArea.Unknown: F_GetTypeName := '<unknown>';
ELSE
	IF NOT F_TcComIecApplicationInfo().GetInterface(ipInterface) THEN RETURN; END_IF
	ipInterface.GetDatatypeNameByAddress(
		TO_UDINT(Variable.diSize), Variable.pValue, nTmp, ADR(F_GetTypeName));
	END_CASE

END_FUNCTION

// ---- POUs/F_TcComIecApplicationInfo.TcPOU
// Provides a reference to a single instance of the FB_TcComIecApplicationInfo function block.
// This function ensures that all parts of the program access the same instance of FB_TcComIecApplicationInfo,
// which can be useful for centralized access to the ITcIecApplicationInfo TcCOM object, resource management, and maintaining consistency.
FUNCTION F_TcComIecApplicationInfo : REFERENCE TO FB_TcComIecApplicationInfo // A reference to an instance of the FB_TcComIecApplicationInfo.
VAR_STAT
	fbTcComIecAppInfo : FB_TcComIecApplicationInfo;
END_VAR

F_TcComIecApplicationInfo REF= fbTcComIecAppInfo;

END_FUNCTION

// ---- POUs/FB_TcComIecApplicationInfo.TcPOU
// Manages the ITcIecApplicationInfo TcCOM Interface.
{attribute 'enable_dynamic_creation'}
{attribute 'no_assign'}
{attribute 'no_explicit_call' := 'direct call for this function block is not allowed'} 
FUNCTION_BLOCK FINAL FB_TcComIecApplicationInfo
VAR
	_ipIecApplicationInformation 	: ITcIecApplicationInfo;
	_hIecApplicationInformation 	: HRESULT := Tc3_Module.GVL.E_FAIL;
END_VAR

{attribute 'hide'}
METHOD FB_exit : BOOL
VAR_INPUT
	bInCopyCode : BOOL; // if TRUE, the exit method is called for exiting an instance that is copied afterwards (online change).
END_VAR
// Return if online change.
IF bInCopyCode THEN RETURN; END_IF

// Safe release of ITcIecApplicationInfo.
Tc3_Module.FW_SafeRelease(ADR(THIS^._ipIecApplicationInformation));
THIS^._hIecApplicationInformation := Tc3_Module.GVL.E_FAIL;
END_METHOD

// Acquires ITcIecApplicationInfo TcCOM interface.
METHOD GetInterface : BOOL // TRUE if the TcCOM interface was successfully acquired.
VAR_IN_OUT
	ipTcComInterface : ITcIecApplicationInfo; // Interface to store acquired TcCOM interface.
END_VAR
// Check if instance already exists. 
// Try to get it of it doesn't.
IF Tc3_Module.FAILED(THIS^._hIecApplicationInformation) THEN
	THIS^._hIecApplicationInformation := Tc3_Module.FW_ObjMgr_GetObjectInstance(
		TwinCAT_SystemInfoVarList._AppInfo.ObjId, 
		TC_GLOBAL_IID_LIST.IID_ITcIecApplicationInfo, 
		ADR(THIS^._ipIecApplicationInformation));
	END_IF

GetInterface 	 := Tc3_Module.SUCCEEDED(THIS^._hIecApplicationInformation);
ipTcComInterface := THIS^._ipIecApplicationInformation;
END_METHOD

END_FUNCTION_BLOCK

// ---- POUs/F_Hash.TcPOU
// Computes a hash value for a given block of memory using the MurmurHash3 algorithm.
// The MurmurHash3 algorithm was created by Austin Appleby. Source: https://en.wikipedia.org/wiki/MurmurHash
FUNCTION F_Hash : DWORD // The computed hash value.
VAR_INPUT
    pAddress 	: POINTER TO BYTE; // The pointer to the beginning of the memory block to be hashed.
    Size 		: T_Size; // The size, in bytes, of the memory block to be hashed.
    Seed 		: DWORD; // A seed value for the hash calculation, which can help in generating different hashes for the same data.
END_VAR
VAR
	i 			: T_Position;
	nK 			: DWORD;
	nBlocks 	: T_Size;
	pBlocks		: POINTER TO DWORD;
	pTail 		: POINTER TO BYTE;
END_VAR
VAR_STAT CONSTANT
	nC1 		: DWORD 			:= 16#CC9E2D51;
	nC2 		: DWORD 			:= 16#1B873593;
END_VAR

IF pAddress = 0 OR Size = 0 THEN RETURN; END_IF

F_Hash := Seed;

nBlocks := Size / 4;
pBlocks := pAddress + nBlocks * 4;

i := -F_SizeToPosition(nBlocks);
FOR i := i TO -1 DO
	nK := pBlocks[i];
	
	nK := nK * nC1;
	nK := SHL(nK, 15) OR SHR(nK, 32 - 15);
	nK := nK * nC2;
	
	F_Hash := F_Hash XOR nK;
	F_Hash := SHL(F_Hash, 13) OR SHR(F_Hash, 32 - 13);
	F_Hash := F_Hash * 5 + 16#E6546B64;
	END_FOR
	
nK := 0;
pTail := pAddress + nBlocks * 4;

i := Size MOD 4;

IF i = 3 THEN 
	{warning disable C0308}
	nK := nK XOR SHL(pTail[2], 16); END_IF;
IF i >= 2 THEN 
	{warning disable C0308}	
	nK := nK XOR SHL(pTail[1], 8); END_IF;
IF i >= 1 THEN
	nK := nK XOR pTail[0];
	nK := nK * nC1;
	nK := SHL(nK, 15) OR SHR(nK, 32 - 15);
	nK := nK * nC2;
	F_Hash := F_Hash XOR nK;
	END_IF;

F_Hash := F_Hash XOR Size;
F_Hash := F_Hash XOR SHR(F_Hash, 16);
F_Hash := F_Hash * 16#85EBCA6B;
F_Hash := F_Hash XOR SHR(F_Hash, 13);
F_Hash := F_Hash * 16#C2B2AE35;
F_Hash := F_Hash XOR SHR(F_Hash, 16);

END_FUNCTION

// ---- POUs/Conversions/F_SizeToPosition.TcPOU
// Converts a size value to a position value.
FUNCTION F_SizeToPosition : T_Position // The position value corresponding to the given size.
VAR_INPUT
	Size : T_Size; // The size value to be converted to a position value.
END_VAR

F_SizeToPosition := Size;

END_FUNCTION

// ---- POUs/P_GetSystemInformation.TcPOU
// Retrieves information about the target.
{attribute 'no_explicit_call' := 'direct call for this program is not allowed'} 
PROGRAM P_GetSystemInformation

// The version as defined in the compile options.
PROPERTY CompilerVersion : VERSION
GET
CompilerVersion := __SYSTEM.Constants.CompilerVersion;
END_GET
END_PROPERTY

// The version as defined in the compile options.
PROPERTY CompilerVersionNumeric : DWORD
GET
CompilerVersionNumeric := __SYSTEM.Constants.CompilerVersionNumeric;
END_GET
END_PROPERTY

// Indicates of whether the target has FPU support.
PROPERTY HasFpuSupport : BOOL
GET
HasFpuSupport := __SYSTEM.Constants.bFPUSupport;
END_GET
END_PROPERTY

// Indicates whether multicore support is available in the target.
PROPERTY HasMulticoreSupport : BOOL
GET
HasMulticoreSupport := __SYSTEM.Constants.bMulticoreSupport;
END_GET
END_PROPERTY

// Indicates if target is in simulation mode.
PROPERTY InSimulationMode : BOOL
GET
InSimulationMode := __SYSTEM.Constants.bSimulationMode;
END_GET
END_PROPERTY

// Indicates of the system is little endian; TRUE for Intel, ARM etc. FALSE for Power PC, etc. 
PROPERTY IsLittleEndian : BOOL
GET
IsLittleEndian := __SYSTEM.Constants.bLittleEndian;
END_GET
END_PROPERTY

// Retrieves the operating system of the target.
PROPERTY OperatingSystem : E_OperatingSystem
GET
VAR_STAT
	nOperatingSystem : UDINT;
	nResult : UDINT := SysTarget.SysTargetGetOperatingSystemId(ADR(nOperatingSystem));
END_VAR
CASE nOperatingSystem OF
	1..4: OperatingSystem := E_OperatingSystem.Windows;
	5: OperatingSystem := E_OperatingSystem.Linux;
	6: OperatingSystem := E_OperatingSystem.VxWorks;
	7: OperatingSystem := E_OperatingSystem.QNX;
	8: OperatingSystem := E_OperatingSystem.uCOS;
ELSE
	OperatingSystem := E_OperatingSystem._;
	END_CASE
END_GET
END_PROPERTY

// Retrieves the packmode of the system.
PROPERTY PackMode : WORD
GET
PackMode := __SYSTEM.Constants.nPackMode;
END_GET
END_PROPERTY

// Retireves the target's processor architecture.
PROPERTY ProcessorArchitecture : E_ProcessorArchitecture
GET
VAR_STAT
	nProcessorArchitecture : UDINT;
	nResult : UDINT := SysTarget.SysTargetGetProcessorId(ADR(nProcessorArchitecture));
END_VAR
ProcessorArchitecture := TO_BYTE(nProcessorArchitecture);
END_GET
END_PROPERTY

// Retrieves the size of the CPU register; 16 for C16x, 64 for X86-64 Bit, 32 for all other controllers.
PROPERTY RegisterSize : WORD
GET
RegisterSize := __SYSTEM.Constants.nRegisterSize;
END_GET
END_PROPERTY

// The version as described in the runtime system.
PROPERTY RuntimeVersion : VERSION
GET
RuntimeVersion := __SYSTEM.Constants.RuntimeVersion;
END_GET
END_PROPERTY

// The version as described in the runtime system.
PROPERTY RuntimeVersionNumeric : DWORD
GET
RuntimeVersionNumeric := __SYSTEM.Constants.RuntimeVersionNumeric;
END_GET
END_PROPERTY

END_PROGRAM

// ---- POUs/F_SetDecimalPlaces.TcPOU
// Sets the specified number of decimal places for a given real value.
FUNCTION F_SetDecimalPlaces : LREAL // The value with the specified number of decimal places.
VAR_INPUT
	fValue 			: LREAL; // The input floating-point value to be rounded.
	nDecimalPlaces 	: USINT; // The number of decimal places to set the number to.
END_VAR

F_SetDecimalPlaces := EXPT(10, nDecimalPlaces);
F_SetDecimalPlaces := 
	LIMIT(
		GVL_TypeValueLimits.LREAL_MIN,
		F_TruncateNumber(fValue * F_SetDecimalPlaces) / F_SetDecimalPlaces,
		GVL_TypeValueLimits.LREAL_MAX);

END_FUNCTION

// ---- POUs/F_TruncateNumber.TcPOU
// Safely retrieves the integer part of a LREAL by truncating the fractional
// component towards zero, without converting to an integer type.
// This avoids PLC crashes caused by casting large LREALs to LINT.
//
// The logic works as follows:
// - For positive numbers: use Tc2_Math.FLOOR(-x) negated → effectively truncates
// - For negative numbers: use Tc2_Math.FLOOR(x) directly → keeps integer part
//
// [Examples]
//  F_TruncateNumber( 3.75 ) →  3.0,
//  F_TruncateNumber(-3.75 ) → -3.0,
//  F_TruncateNumber( 0.99 ) →  0.0,
//  F_TruncateNumber(-0.99 ) →  0.0,
//  F_TruncateNumber( 1.7e+308 ) → 1.7e+308 (no crash)
//
// This function is a safe alternative to TRUNC() or Tc2_Math.TRUNC(), especially
// for edge cases near the limits of the LREAL type.
FUNCTION F_TruncateNumber : LREAL // The integer part of a LREAL by truncating the fractional component towards zero.
VAR_INPUT
	fValue : LREAL; // The input floating-point value to truncate
END_VAR

F_TruncateNumber :=
	SEL(fValue < 0, Tc2_Math.FLOOR(fValue), -Tc2_Math.FLOOR(-fValue));

END_FUNCTION

// ---- POUs/F_SearchMemory.TcPOU
// Searches for a specific sequence of bytes in a given memory area.
FUNCTION F_SearchMemory : POINTER TO BYTE // Pointer to the start of the found sequence, or 0 if not found.
VAR_INPUT
    pAddress    : POINTER TO BYTE; // Starting address of the memory area to search.
    Size 		: T_Size; // Size of the memory area (in bytes).
    pValue   	: POINTER TO BYTE; // Pointer to the sequence of bytes to search for.
    ValueSize	: T_Size; // Size of the sequence of bytes (in bytes).
END_VAR
VAR_OUTPUT
	Index		: T_Position := -1; // Index of the start of the found sequence, or -1 if not found.
END_VAR
VAR
    i, j,
	iEnd, jEnd	: T_Position;
END_VAR

IF pAddress = 0 OR pValue = 0 OR ValueSize = 0 THEN RETURN; END_IF

iEnd := F_SizeToPosition(Size) - ValueSize;
jEnd := F_SizeToPosition(ValueSize) - 1;
FOR i := 0 TO iEnd DO
	FOR j := 0 TO jEnd DO
		IF pAddress[i + j] <> pValue[j] THEN EXIT; END_IF
		END_FOR
	IF j = ValueSize THEN F_SearchMemory := ADR(pAddress[i]); Index := j; RETURN; END_IF
	END_FOR

END_FUNCTION

// ---- POUs/Conversions/F_IntToSize.TcPOU
// Converts a INT value to a size value, ensuring it falls within the defined limits.
FUNCTION F_IntToSize : T_Size // The size value constrained within the minimum and maximum limits of T_Size.
VAR_INPUT
	nValue : INT; // The INT value to be converted to a size value.
END_VAR
VAR
END_VAR

F_IntToSize := TO_UDINT(
	LIMIT(0, nValue, GVL_TypeValueLimits.INT_MAX));

END_FUNCTION

// ---- POUs/F_ResetOnTrue.TcPOU
// Sets the boolean value to false if it is true and returns true if it was true before being set.
FUNCTION F_ResetOnTrue : BOOL // Whether the value was true before resetting.
VAR_INPUT
	bValue : REFERENCE TO BOOL; // Boolean value to reset.
END_VAR

F_ResetOnTrue 	:= bValue;
bValue 			:= FALSE;

END_FUNCTION

// ---- POUs/Bounds/F_GetBoolArrayUpperBound.TcPOU
// Gets the upper bound index of the array of specified type.
FUNCTION F_GetBoolArrayUpperBound : T_Position // The upper bound index of the specified array.
VAR_IN_OUT
	arArray : ARRAY[*] OF BOOL; // The array to query.
END_VAR

F_GetBoolArrayUpperBound := UPPER_BOUND(arArray, 1);

END_FUNCTION

// ---- POUs/Bounds/F_GetByteArrayUpperBound.TcPOU
// Gets the upper bound index of the array of specified type.
FUNCTION F_GetByteArrayUpperBound : T_Position // The upper bound index of the specified array.
VAR_IN_OUT
	arArray : ARRAY[*] OF BYTE; // The array to query.
END_VAR

F_GetByteArrayUpperBound := UPPER_BOUND(arArray, 1);

END_FUNCTION

// ---- POUs/Bounds/F_GetDateAndTimeArrayUpperBound.TcPOU
// Gets the upper bound index of the array of specified type.
FUNCTION F_GetDateAndTimeArrayUpperBound : T_Position // The upper bound index of the specified array.
VAR_IN_OUT
	arArray : ARRAY[*] OF DATE_AND_TIME; // The array to query.
END_VAR

F_GetDateAndTimeArrayUpperBound := UPPER_BOUND(arArray, 1);

END_FUNCTION

// ---- POUs/Bounds/F_GetDateArrayUpperBound.TcPOU
// Gets the upper bound index of the array of specified type.
FUNCTION F_GetDateArrayUpperBound : T_Position // The upper bound index of the specified array.
VAR_IN_OUT
	arArray : ARRAY[*] OF DATE; // The array to query.
END_VAR

F_GetDateArrayUpperBound := UPPER_BOUND(arArray, 1);

END_FUNCTION

// ---- POUs/Bounds/F_GetDIntArrayUpperBound.TcPOU
// Gets the upper bound index of the array of specified type.
FUNCTION F_GetDIntArrayUpperBound : T_Position // The upper bound index of the specified array.
VAR_IN_OUT
	arArray : ARRAY[*] OF DINT; // The array to query.
END_VAR

F_GetDIntArrayUpperBound := UPPER_BOUND(arArray, 1);

END_FUNCTION

// ---- POUs/Bounds/F_GetDWordArrayUpperBound.TcPOU
// Gets the upper bound index of the array of specified type.
FUNCTION F_GetDWordArrayUpperBound : T_Position // The upper bound index of the specified array.
VAR_IN_OUT
	arArray : ARRAY[*] OF DWORD; // The array to query.
END_VAR

F_GetDWordArrayUpperBound := UPPER_BOUND(arArray, 1);

END_FUNCTION

// ---- POUs/Bounds/F_GetIntArrayUpperBound.TcPOU
// Gets the upper bound index of the array of specified type.
FUNCTION F_GetIntArrayUpperBound : T_Position // The upper bound index of the specified array.
VAR_IN_OUT
	arArray : ARRAY[*] OF INT; // The array to query.
END_VAR

F_GetIntArrayUpperBound := UPPER_BOUND(arArray, 1);

END_FUNCTION

// ---- POUs/Bounds/F_GetInterfaceArrayLowerBound.TcPOU
// Gets the lower bound index of the array of specified type.
FUNCTION F_GetInterfaceArrayLowerBound : T_Position // The lower bound index of the specified array.
VAR_IN_OUT
	arArray : ARRAY[*] OF __SYSTEM.IQueryInterface; // The array to query.
END_VAR

F_GetInterfaceArrayLowerBound := LOWER_BOUND(arArray, 1);

END_FUNCTION

// ---- POUs/Bounds/F_GetInterfaceArrayUpperBound.TcPOU
// Gets the upper bound index of the array of specified type.
FUNCTION F_GetInterfaceArrayUpperBound : T_Position // The upper bound index of the specified array.
VAR_IN_OUT
	arArray : ARRAY[*] OF __SYSTEM.IQueryInterface; // The array to query.
END_VAR

F_GetInterfaceArrayUpperBound := UPPER_BOUND(arArray, 1);

END_FUNCTION

// ---- POUs/Bounds/F_GetLIntArrayUpperBound.TcPOU
// Gets the upper bound index of the array of specified type.
FUNCTION F_GetLIntArrayUpperBound : T_Position // The upper bound index of the specified array.
VAR_IN_OUT
	arArray : ARRAY[*] OF LINT; // The array to query.
END_VAR

F_GetLIntArrayUpperBound := UPPER_BOUND(arArray, 1);

END_FUNCTION

// ---- POUs/Bounds/F_GetLRealArrayUpperBound.TcPOU
// Gets the upper bound index of the array of specified type.
FUNCTION F_GetLRealArrayUpperBound : T_Position // The upper bound index of the specified array.
VAR_IN_OUT
	arArray : ARRAY[*] OF LREAL; // The array to query.
END_VAR

F_GetLRealArrayUpperBound := UPPER_BOUND(arArray, 1);

END_FUNCTION

// ---- POUs/Bounds/F_GetLTimeArrayUpperBound.TcPOU
// Gets the upper bound index of the array of specified type.
FUNCTION F_GetLTimeArrayUpperBound : T_Position // The upper bound index of the specified array.
VAR_IN_OUT
	arArray : ARRAY[*] OF LTIME; // The array to query.
END_VAR

F_GetLTimeArrayUpperBound := UPPER_BOUND(arArray, 1);

END_FUNCTION

// ---- POUs/Bounds/F_GetLWordArrayUpperBound.TcPOU
// Gets the upper bound index of the array of specified type.
FUNCTION F_GetLWordArrayUpperBound : T_Position // The upper bound index of the specified array.
VAR_IN_OUT
	arArray : ARRAY[*] OF LWORD; // The array to query.
END_VAR

F_GetLWordArrayUpperBound := UPPER_BOUND(arArray, 1);

END_FUNCTION

// ---- POUs/Bounds/F_GetMaxStringArrayLowerBound.TcPOU
// Gets the lower bound index of the array of specified type.
FUNCTION F_GetMaxStringArrayLowerBound : T_Position // The lower bound index of the specified array.
VAR_IN_OUT
	arArray : ARRAY[*] OF Tc2_System.T_MaxString; // The array to query.
END_VAR

F_GetMaxStringArrayLowerBound := LOWER_BOUND(arArray, 1);

END_FUNCTION

// ---- POUs/Bounds/F_GetMaxStringArrayUpperBound.TcPOU
// Gets the upper bound index of the array of specified type.
FUNCTION F_GetMaxStringArrayUpperBound : T_Position // The upper bound index of the specified array.
VAR_IN_OUT
	arArray : ARRAY[*] OF Tc2_System.T_MaxString; // The array to query.
END_VAR

F_GetMaxStringArrayUpperBound := UPPER_BOUND(arArray, 1);

END_FUNCTION

// ---- POUs/Bounds/F_GetMaxWStringArrayLowerBound.TcPOU
// Gets the lower bound index of the array of specified type.
FUNCTION F_GetMaxWStringArrayLowerBound : T_Position // The lower bound index of the specified array.
VAR_IN_OUT
	arArray : ARRAY[*] OF T_MaxWString; // The array to query.
END_VAR

F_GetMaxWStringArrayLowerBound := LOWER_BOUND(arArray, 1);

END_FUNCTION

// ---- POUs/Bounds/F_GetMaxWStringArrayUpperBound.TcPOU
// Gets the upper bound index of the array of specified type.
FUNCTION F_GetMaxWStringArrayUpperBound : T_Position // The upper bound index of the specified array.
VAR_IN_OUT
	arArray : ARRAY[*] OF T_MaxWString; // The array to query.
END_VAR

F_GetMaxWStringArrayUpperBound := UPPER_BOUND(arArray, 1);

END_FUNCTION

// ---- POUs/Bounds/F_GetPointerArrayUpperBound.TcPOU
// Gets the upper bound index of the array of specified type.
FUNCTION F_GetPointerArrayUpperBound : T_Position // The upper bound index of the specified array.
VAR_IN_OUT
	arArray : ARRAY[*] OF POINTER TO BYTE; // The array to query.
END_VAR

F_GetPointerArrayUpperBound := UPPER_BOUND(arArray, 1);

END_FUNCTION

// ---- POUs/Bounds/F_GetRealArrayUpperBound.TcPOU
// Gets the upper bound index of the array of specified type.
FUNCTION F_GetRealArrayUpperBound : T_Position // The upper bound index of the specified array.
VAR_IN_OUT
	arArray : ARRAY[*] OF REAL; // The array to query.
END_VAR

F_GetRealArrayUpperBound := UPPER_BOUND(arArray, 1);

END_FUNCTION

// ---- POUs/Bounds/F_GetRunnableArrayLowerBound.TcPOU
(* Gets the lower bound index of :itf:`I_Runnable` array.*)
FUNCTION F_GetRunnableArrayLowerBound : T_Position
VAR_IN_OUT
	arRunnables : ARRAY[*] OF REAL; // The array to query.
END_VAR

F_GetRunnableArrayLowerBound := LOWER_BOUND(arRunnables, 1);

END_FUNCTION

// ---- POUs/Bounds/F_GetRunnableArrayUpperBound.TcPOU
(* Gets the upper bound index of :itf:`I_Runnable` array.*)
FUNCTION F_GetRunnableArrayUpperBound : T_Position
VAR_IN_OUT
	arRunnables : ARRAY[*] OF REAL; // The array to query.
END_VAR

F_GetRunnableArrayUpperBound := LOWER_BOUND(arRunnables, 1);

END_FUNCTION

// ---- POUs/Bounds/F_GetSIntArrayUpperBound.TcPOU
// Gets the upper bound index of the array of specified type.
FUNCTION F_GetSIntArrayUpperBound : T_Position // The upper bound index of the specified array.
VAR_IN_OUT
	arArray : ARRAY[*] OF SINT; // The array to query.
END_VAR

F_GetSIntArrayUpperBound := UPPER_BOUND(arArray, 1);

END_FUNCTION

// ---- POUs/Bounds/F_GetStringArrayUpperBound.TcPOU
// Gets the upper bound index of the array of specified type.
FUNCTION F_GetStringArrayUpperBound : T_Position // The upper bound index of the specified array.
VAR_IN_OUT
	arArray : ARRAY[*] OF STRING; // The array to query.
END_VAR

F_GetStringArrayUpperBound := UPPER_BOUND(arArray, 1);

END_FUNCTION

// ---- POUs/Bounds/F_GetTimeArrayUpperBound.TcPOU
// Gets the upper bound index of the array of specified type.
FUNCTION F_GetTimeArrayUpperBound : T_Position // The upper bound index of the specified array.
VAR_IN_OUT
	arArray : ARRAY[*] OF TIME; // The array to query.
END_VAR

F_GetTimeArrayUpperBound := UPPER_BOUND(arArray, 1);

END_FUNCTION

// ---- POUs/Bounds/F_GetTimeOfDayArrayUpperBound.TcPOU
// Gets the upper bound index of the array of specified type.
FUNCTION F_GetTimeOfDayArrayUpperBound : T_Position // The upper bound index of the specified array.
VAR_IN_OUT
	arArray : ARRAY[*] OF TIME_OF_DAY; // The array to query.
END_VAR

F_GetTimeOfDayArrayUpperBound := UPPER_BOUND(arArray, 1);

END_FUNCTION

// ---- POUs/Bounds/F_GetUDIntArrayUpperBound.TcPOU
// Gets the upper bound index of the array of specified type.
FUNCTION F_GetUDIntArrayUpperBound : T_Position // The upper bound index of the specified array.
VAR_IN_OUT
	arArray : ARRAY[*] OF UDINT; // The array to query.
END_VAR

F_GetUDIntArrayUpperBound := UPPER_BOUND(arArray, 1);

END_FUNCTION

// ---- POUs/Bounds/F_GetUIntArrayUpperBound.TcPOU
// Gets the upper bound index of the array of specified type.
FUNCTION F_GetUIntArrayUpperBound : T_Position // The upper bound index of the specified array.
VAR_IN_OUT
	arArray : ARRAY[*] OF UINT; // The array to query.
END_VAR

F_GetUIntArrayUpperBound := UPPER_BOUND(arArray, 1);

END_FUNCTION

// ---- POUs/Bounds/F_GetULIntArrayUpperBound.TcPOU
// Gets the upper bound index of the array of specified type.
FUNCTION F_GetULIntArrayUpperBound : T_Position // The upper bound index of the specified array.
VAR_IN_OUT
	arArray : ARRAY[*] OF ULINT; // The array to query.
END_VAR

F_GetULIntArrayUpperBound := UPPER_BOUND(arArray, 1);

END_FUNCTION

// ---- POUs/Bounds/F_GetUSIntArrayUpperBound.TcPOU
// Gets the upper bound index of the array of specified type.
FUNCTION F_GetUSIntArrayUpperBound : T_Position // The upper bound index of the specified array.
VAR_IN_OUT
	arArray : ARRAY[*] OF USINT; // The array to query.
END_VAR

F_GetUSIntArrayUpperBound := UPPER_BOUND(arArray, 1);

END_FUNCTION

// ---- POUs/Bounds/F_GetUXIntArrayUpperBound.TcPOU
// Gets the upper bound index of the array of specified type.
FUNCTION F_GetUXIntArrayUpperBound : T_Position // The upper bound index of the specified array.
VAR_IN_OUT
	arArray : ARRAY[*] OF __UXINT; // The array to query.
END_VAR

F_GetUXIntArrayUpperBound := UPPER_BOUND(arArray, 1);

END_FUNCTION

// ---- POUs/Bounds/F_GetWordArrayUpperBound.TcPOU
// Gets the upper bound index of the array of specified type.
FUNCTION F_GetWordArrayUpperBound : T_Position // The upper bound index of the specified array.
VAR_IN_OUT
	arArray : ARRAY[*] OF WORD; // The array to query.
END_VAR

F_GetWordArrayUpperBound := UPPER_BOUND(arArray, 1);

END_FUNCTION

// ---- POUs/Bounds/F_GetWStringArrayLowerBound.TcPOU
// Gets the lower bound index of the array of specified type.
FUNCTION F_GetWStringArrayLowerBound : T_Position // The lower bound index of the specified array.
VAR_IN_OUT
	arArray : ARRAY[*] OF WSTRING; // The array to query.
END_VAR

F_GetWStringArrayLowerBound := LOWER_BOUND(arArray, 1);

END_FUNCTION

// ---- POUs/Bounds/F_GetStringArrayLowerBound.TcPOU
// Gets the lower bound index of the array of specified type.
FUNCTION F_GetStringArrayLowerBound : T_Position // The lower bound index of the specified array.
VAR_IN_OUT
	arArray : ARRAY[*] OF STRING; // The array to query.
END_VAR

F_GetStringArrayLowerBound := LOWER_BOUND(arArray, 1);

END_FUNCTION

// ---- POUs/Bounds/F_GetPointerArrayLowerBound.TcPOU
// Gets the lower bound index of the array of specified type.
FUNCTION F_GetPointerArrayLowerBound : T_Position // The lower bound index of the specified array.
VAR_IN_OUT
	arArray : ARRAY[*] OF POINTER TO BYTE; // The array to query.
END_VAR

F_GetPointerArrayLowerBound := LOWER_BOUND(arArray, 1);

END_FUNCTION

// ---- POUs/Bounds/F_GetTimeOfDayArrayLowerBound.TcPOU
// Gets the lower bound index of the array of specified type.
FUNCTION F_GetTimeOfDayArrayLowerBound : T_Position // The lower bound index of the specified array.
VAR_IN_OUT
	arArray : ARRAY[*] OF TIME_OF_DAY; // The array to query.
END_VAR

F_GetTimeOfDayArrayLowerBound := LOWER_BOUND(arArray, 1);

END_FUNCTION

// ---- POUs/Bounds/F_GetDateAndTimeArrayLowerBound.TcPOU
// Gets the lower bound index of the array of specified type.
FUNCTION F_GetDateAndTimeArrayLowerBound : T_Position // The lower bound index of the specified array.
VAR_IN_OUT
	arArray : ARRAY[*] OF DATE_AND_TIME; // The array to query.
END_VAR

F_GetDateAndTimeArrayLowerBound := LOWER_BOUND(arArray, 1);

END_FUNCTION

// ---- POUs/Bounds/F_GetDateArrayLowerBound.TcPOU
// Gets the lower bound index of the array of specified type.
FUNCTION F_GetDateArrayLowerBound : T_Position // The lower bound index of the specified array.
VAR_IN_OUT
	arArray : ARRAY[*] OF DATE; // The array to query.
END_VAR

F_GetDateArrayLowerBound := LOWER_BOUND(arArray, 1);

END_FUNCTION

// ---- POUs/Bounds/F_GetTimeArrayLowerBound.TcPOU
// Gets the lower bound index of the array of specified type.
FUNCTION F_GetTimeArrayLowerBound : T_Position // The lower bound index of the specified array.
VAR_IN_OUT
	arArray : ARRAY[*] OF TIME; // The array to query.
END_VAR

F_GetTimeArrayLowerBound := LOWER_BOUND(arArray, 1);

END_FUNCTION

// ---- POUs/Bounds/F_GetRealArrayLowerBound.TcPOU
// Gets the lower bound index of the array of specified type.
FUNCTION F_GetRealArrayLowerBound : T_Position // The lower bound index of the specified array.
VAR_IN_OUT
	arArray : ARRAY[*] OF REAL; // The array to query.
END_VAR

F_GetRealArrayLowerBound := LOWER_BOUND(arArray, 1);

END_FUNCTION

// ---- POUs/Bounds/F_GetLRealArrayLowerBound.TcPOU
// Gets the lower bound index of the array of specified type.
FUNCTION F_GetLRealArrayLowerBound : T_Position // The lower bound index of the specified array.
VAR_IN_OUT
	arArray : ARRAY[*] OF LREAL; // The array to query.
END_VAR

F_GetLRealArrayLowerBound := LOWER_BOUND(arArray, 1);

END_FUNCTION

// ---- POUs/Bounds/F_GetLTimeArrayLowerBound.TcPOU
// Gets the lower bound index of the array of specified type.
FUNCTION F_GetLTimeArrayLowerBound : T_Position // The lower bound index of the specified array.
VAR_IN_OUT
	arArray : ARRAY[*] OF LTIME; // The array to query.
END_VAR

F_GetLTimeArrayLowerBound := LOWER_BOUND(arArray, 1);

END_FUNCTION

// ---- POUs/Bounds/F_GetUDIntArrayLowerBound.TcPOU
// Gets the lower bound index of the array of specified type.
FUNCTION F_GetUDIntArrayLowerBound : T_Position // The lower bound index of the specified array.
VAR_IN_OUT
	arArray : ARRAY[*] OF UDINT; // The array to query.
END_VAR

F_GetUDIntArrayLowerBound := LOWER_BOUND(arArray, 1);

END_FUNCTION

// ---- POUs/Bounds/F_GetULIntArrayLowerBound.TcPOU
// Gets the lower bound index of the array of specified type.
FUNCTION F_GetULIntArrayLowerBound : T_Position // The lower bound index of the specified array.
VAR_IN_OUT
	arArray : ARRAY[*] OF ULINT; // The array to query.
END_VAR

F_GetULIntArrayLowerBound := LOWER_BOUND(arArray, 1);

END_FUNCTION

// ---- POUs/Bounds/F_GetUXIntArrayLowerBound.TcPOU
// Gets the lower bound index of the array of specified type.
FUNCTION F_GetUXIntArrayLowerBound : T_Position // The lower bound index of the specified array.
VAR_IN_OUT
	arArray : ARRAY[*] OF __UXINT; // The array to query.
END_VAR

F_GetUXIntArrayLowerBound := LOWER_BOUND(arArray, 1);

END_FUNCTION

// ---- POUs/Bounds/F_GetUSIntArrayLowerBound.TcPOU
// Gets the lower bound index of the array of specified type.
FUNCTION F_GetUSIntArrayLowerBound : T_Position // The lower bound index of the specified array.
VAR_IN_OUT
	arArray : ARRAY[*] OF USINT; // The array to query.
END_VAR

F_GetUSIntArrayLowerBound := LOWER_BOUND(arArray, 1);

END_FUNCTION

// ---- POUs/Bounds/F_GetDIntArrayLowerBound.TcPOU
// Gets the lower bound index of the array of specified type.
FUNCTION F_GetDIntArrayLowerBound : T_Position // The lower bound index of the specified array.
VAR_IN_OUT
	arArray : ARRAY[*] OF DINT; // The array to query.
END_VAR

F_GetDIntArrayLowerBound := LOWER_BOUND(arArray, 1);

END_FUNCTION

// ---- POUs/Bounds/F_GetLIntArrayLowerBound.TcPOU
// Gets the lower bound index of the array of specified type.
FUNCTION F_GetLIntArrayLowerBound : T_Position // The lower bound index of the specified array.
VAR_IN_OUT
	arArray : ARRAY[*] OF LINT; // The array to query.
END_VAR

F_GetLIntArrayLowerBound := LOWER_BOUND(arArray, 1);

END_FUNCTION

// ---- POUs/Bounds/F_GetUIntArrayLowerBound.TcPOU
// Gets the lower bound index of the array of specified type.
FUNCTION F_GetUIntArrayLowerBound : T_Position // The lower bound index of the specified array.
VAR_IN_OUT
	arArray : ARRAY[*] OF UINT; // The array to query.
END_VAR

F_GetUIntArrayLowerBound := LOWER_BOUND(arArray, 1);

END_FUNCTION

// ---- POUs/Bounds/F_GetWStringArrayUpperBound.TcPOU
// Gets the upper bound index of the array of specified type.
FUNCTION F_GetWStringArrayUpperBound : T_Position // The upper bound index of the specified array.
VAR_IN_OUT
	arArray : ARRAY[*] OF WSTRING; // The array to query.
END_VAR

F_GetWStringArrayUpperBound := UPPER_BOUND(arArray, 1);

END_FUNCTION

// ---- POUs/Bounds/F_GetXIntArrayLowerBound.TcPOU
// Gets the lower bound index of the array of specified type.
FUNCTION F_GetXIntArrayLowerBound : T_Position // The lower bound index of the specified array.
VAR_IN_OUT
	arArray : ARRAY[*] OF __XINT; // The array to query.
END_VAR

F_GetXIntArrayLowerBound := LOWER_BOUND(arArray, 1);

END_FUNCTION

// ---- POUs/Bounds/F_GetSIntArrayLowerBound.TcPOU
// Gets the lower bound index of the array of specified type.
FUNCTION F_GetSIntArrayLowerBound : T_Position // The lower bound index of the specified array.
VAR_IN_OUT
	arArray : ARRAY[*] OF SINT; // The array to query.
END_VAR

F_GetSIntArrayLowerBound := LOWER_BOUND(arArray, 1);

END_FUNCTION

// ---- POUs/Bounds/F_GetByteArrayLowerBound.TcPOU
// Gets the lower bound index of the array of specified type.
FUNCTION F_GetByteArrayLowerBound : T_Position // The lower bound index of the specified array.
VAR_IN_OUT
	arArray : ARRAY[*] OF BYTE; // The array to query.
END_VAR

F_GetByteArrayLowerBound := LOWER_BOUND(arArray, 1);

END_FUNCTION

// ---- POUs/Bounds/F_GetBoolArrayLowerBound.TcPOU
// Gets the lower bound index of the array of specified type.
FUNCTION F_GetBoolArrayLowerBound : T_Position // The lower bound index of the specified array.
VAR_IN_OUT
	arArray : ARRAY[*] OF BOOL; // The array to query.
END_VAR

F_GetBoolArrayLowerBound := LOWER_BOUND(arArray, 1);

END_FUNCTION

// ---- POUs/Bounds/F_GetLWordArrayLowerBound.TcPOU
// Gets the lower bound index of the array of specified type.
FUNCTION F_GetLWordArrayLowerBound : T_Position // The lower bound index of the specified array.
VAR_IN_OUT
	arArray : ARRAY[*] OF LWORD; // The array to query.
END_VAR

F_GetLWordArrayLowerBound := LOWER_BOUND(arArray, 1);

END_FUNCTION

// ---- POUs/Bounds/F_GetIntArrayLowerBound.TcPOU
// Gets the lower bound index of the array of specified type.
FUNCTION F_GetIntArrayLowerBound : T_Position // The lower bound index of the specified array.
VAR_IN_OUT
	arArray : ARRAY[*] OF INT; // The array to query.
END_VAR

F_GetIntArrayLowerBound := LOWER_BOUND(arArray, 1);

END_FUNCTION

// ---- POUs/Bounds/F_GetXIntArrayUpperBound.TcPOU
// Gets the upper bound index of the array of specified type.
FUNCTION F_GetXIntArrayUpperBound : T_Position // The upper bound index of the specified array.
VAR_IN_OUT
	arArray : ARRAY[*] OF __XINT; // The array to query.
END_VAR

F_GetXIntArrayUpperBound := UPPER_BOUND(arArray, 1);

END_FUNCTION

// ---- POUs/Bounds/F_GetXWordArrayLowerBound.TcPOU
// Gets the lower bound index of the array of specified type.
FUNCTION F_GetXWordArrayLowerBound : T_Position // The lower bound index of the specified array.
VAR_IN_OUT
	arArray : ARRAY[*] OF __XWORD; // The array to query.
END_VAR

F_GetXWordArrayLowerBound := LOWER_BOUND(arArray, 1);

END_FUNCTION

// ---- POUs/Bounds/F_GetWordArrayLowerBound.TcPOU
// Gets the lower bound index of the array of specified type.
FUNCTION F_GetWordArrayLowerBound : T_Position // The lower bound index of the specified array.
VAR_IN_OUT
	arArray : ARRAY[*] OF WORD; // The array to query.
END_VAR

F_GetWordArrayLowerBound := LOWER_BOUND(arArray, 1);

END_FUNCTION

// ---- POUs/Bounds/F_GetDWordArrayLowerBound.TcPOU
// Gets the lower bound index of the array of specified type.
FUNCTION F_GetDWordArrayLowerBound : T_Position // The lower bound index of the specified array.
VAR_IN_OUT
	arArray : ARRAY[*] OF DWORD; // The array to query.
END_VAR

F_GetDWordArrayLowerBound := LOWER_BOUND(arArray, 1);

END_FUNCTION

// ---- POUs/Bounds/F_GetXWordArrayUpperBound.TcPOU
// Gets the upper bound index of the array of specified type.
FUNCTION F_GetXWordArrayUpperBound : T_Position // The upper bound index of the specified array.
VAR_IN_OUT
	arArray : ARRAY[*] OF __XWORD; // The array to query.
END_VAR

F_GetXWordArrayUpperBound := UPPER_BOUND(arArray, 1);

END_FUNCTION

// ---- POUs/Conversions/F_DintToSize.TcPOU
// Converts a DINT value to a size value, ensuring it falls within the defined limits.
FUNCTION F_DintToSize : T_Size // The size value constrained within the minimum and maximum limits of T_Size.
VAR_INPUT
	nValue : DINT; // The DINT value to be converted to a size value.
END_VAR
VAR
END_VAR

F_DintToSize := TO_UDINT(
	LIMIT(0, nValue, GVL_TypeValueLimits.DINT_MAX));

END_FUNCTION

// ---- POUs/Conversions/F_ULintToPosition.TcPOU
// Converts a ULINT value to a position value, ensuring it falls within the defined limits.
FUNCTION F_ULintToPosition : T_Position // The position value constrained within the minimum and maximum limits of T_Position.
VAR_INPUT
	nValue : ULINT; // The size value to be converted to a position value.
END_VAR

F_ULintToPosition := TO_LINT(LIMIT(0, nValue, TO_ULINT(GVL_TypeValueLimits.LINT_MAX)));

END_FUNCTION

// ---- POUs/FB_ValueChangeDetector.TcPOU
// Detects if the watched variable value has changed.
{attribute 'enable_dynamic_creation'}
FUNCTION_BLOCK FINAL FB_ValueChangeDetector IMPLEMENTS I_ChangeDetector
VAR_INPUT
	Value : ANY; // Value to detect for change.
END_VAR
VAR
	_nHash : DWORD;
END_VAR

// Indicates if the value has changed.
// [get] Returns flag indicating of value has changed.
PROPERTY HasChanged : BOOL
GET
VAR_INST
	bFirstCall : BOOL := TRUE;
END_VAR
VAR
	nHash : DWORD;
END_VAR
nHash := F_Hash(THIS^.Value.pValue,
				F_PositionToSize(THIS^.Value.diSize),
				THIS^.Value.TypeClass);

HasChanged := THIS^._nHash <> nHash OR_ELSE F_ResetOnTrue(bFirstCall);

IF HasChanged THEN THIS^._nHash := nHash; END_IF
END_GET
END_PROPERTY

END_FUNCTION_BLOCK

// ---- POUs/F_AllAreFalse.TcPOU
// Checks if all elements in a boolean array are false.
FUNCTION F_AllAreFalse : BOOL // True if all elements in the array are false.
VAR_IN_OUT
	arValues : ARRAY[*] OF BOOL; // An array of boolean values to check.
END_VAR
VAR
	i : T_Position;
END_VAR

FOR i := LOWER_BOUND(arValues, 1) TO UPPER_BOUND(arValues, 1) DO
	IF arValues[i] THEN RETURN; END_IF 
	END_FOR
	
F_AllAreFalse := TRUE;

END_FUNCTION

// ---- POUs/F_AllocateMemory.TcPOU
// Allocates a block of dynamic memory of the specified size.
FUNCTION F_AllocateMemory : POINTER TO BYTE // A pointer to the beginning of the newly allocated memory block.
VAR_INPUT
	Size : T_Size; // The size, in bytes, of the memory block to be allocated.
END_VAR

F_AllocateMemory := __NEW(BYTE, Size);

END_FUNCTION

// ---- POUs/F_AnyAreTrue.TcPOU
// Checks if any element in a boolean array is true.
FUNCTION F_AnyAreTrue : BOOL // True if any element in the array is true.
VAR_IN_OUT
	arValues : ARRAY[*] OF BOOL; // An array of boolean values to check.
END_VAR
VAR
	i : T_Position;
END_VAR

FOR i := LOWER_BOUND(arValues, 1) TO UPPER_BOUND(arValues, 1) DO
	IF arValues[i] THEN F_AnyAreTrue := TRUE; RETURN; END_IF 
	END_FOR

END_FUNCTION

// ---- POUs/F_AnyAreFalse.TcPOU
// Checks if any element in a boolean array is false.
FUNCTION F_AnyAreFalse : BOOL // True if any element in the array is false.
VAR_IN_OUT
	arValues : ARRAY[*] OF BOOL; // An array of boolean values to check.
END_VAR
VAR
	i : T_Position;
END_VAR

FOR i := LOWER_BOUND(arValues, 1) TO UPPER_BOUND(arValues, 1) DO
	IF NOT arValues[i] THEN F_AnyAreFalse := TRUE; RETURN; END_IF 
	END_FOR

END_FUNCTION

// ---- POUs/F_AreSameTypeFromInterfaces.TcPOU
// Checks if both interfaces come from the same concrete FB type.
FUNCTION F_AreSameTypeFromInterfaces : BOOL // TRUE if supplied interfaces are from the same concrete type.
VAR_INPUT
	// Interface to compare.
	ipA	: __SYSTEM.IQueryInterface;
	// Interface to compare.
	ipB : __SYSTEM.IQueryInterface;
END_VAR
VAR
	pA, pB : POINTER TO __UXINT;
END_VAR

pA := F_GetAddressFromInterface(ipA);
pB := F_GetAddressFromInterface(ipB);

F_AreSameTypeFromInterfaces := (pA <> 0 AND pB <> 0) AND_THEN pA^ = pB^;

END_FUNCTION

// ---- POUs/F_GetAddressFromInterface.TcPOU
// Retrieves the memory address of an object given its interface.
FUNCTION F_GetAddressFromInterface : POINTER TO BYTE // A pointer to the memory address of the object corresponding to the provided interface pointer.
VAR_INPUT
	ipInterface : __SYSTEM.IQueryInterface; // The interface from which the address of the object will be extracted.
END_VAR
VAR
	pInterface : POINTER TO POINTER TO BYTE := ADR(ipInterface);
END_VAR

F_GetAddressFromInterface := SEL(ipInterface <> 0, 0, pInterface^ - SIZEOF(ipInterface));

END_FUNCTION

// ---- POUs/F_ExtractPointerFromInterface.TcPOU
// Extracts the underlying object pointer from an interface pointer.
// [note] The interface must inherit from __SYSTEM.IQueryInterface, otherwise the check is not valid.
FUNCTION F_ExtractPointerFromInterface : POINTER TO BYTE // Returns pointer to the concrete object or 0 if invalid.
VAR_INPUT
	// Address of the interface (e.g. ADR(ipInterface)).
	pInterface : POINTER TO BYTE;
END_VAR
VAR
	pTmp : POINTER TO POINTER TO BYTE := pInterface;
END_VAR

RETURN( NOT(F_IsReadablePointer(pInterface) AND F_IsPointerToInterface(pInterface)) );

F_ExtractPointerFromInterface := pTmp^;

END_FUNCTION

// ---- POUs/F_IsReadablePointer.TcPOU
// Checks if a pointer is in a readable memory area (static/dynamic).
FUNCTION F_IsReadablePointer : BOOL // TRUE if the given pointer refers to a readable memory area.
VAR_INPUT
	// Pointer to check for readability.
	pValue : POINTER TO BYTE;
END_VAR
VAR
END_VAR

RETURN(pValue = 0);

CASE F_GetAddressMemoryArea(pValue) OF 
	E_AddressMemoryArea.Static,
	E_AddressMemoryArea.Dynamic:
		F_IsReadablePointer := TRUE;
	END_CASE

END_FUNCTION

// ---- POUs/F_GetAddressMemoryArea.TcPOU
// Determines the memory area type of a given pointer.
FUNCTION F_GetAddressMemoryArea : E_AddressMemoryArea // An enumeration indicating the type of memory area the address belongs to.
VAR_INPUT
	pAddress : POINTER TO BYTE; // The memory address pointer to be checked.
END_VAR

CASE Tc2_System.F_CheckMemoryArea(pAddress, 1) OF
	Tc2_System.E_TcMemoryArea.Static:	F_GetAddressMemoryArea := E_AddressMemoryArea.Static;
	Tc2_System.E_TcMemoryArea.Dynamic:	F_GetAddressMemoryArea := E_AddressMemoryArea.Dynamic;
	Tc2_System.E_TcMemoryArea.CNC:		F_GetAddressMemoryArea := E_AddressMemoryArea.CNC;
ELSE
	F_GetAddressMemoryArea := E_AddressMemoryArea._;
	END_CASE

END_FUNCTION

// ---- POUs/F_IsPointerToInterface.TcPOU
// Tries to guess if the given pointer refers to an interface instance.
// [note]
// This is heuristic and can be inaccurate. The object MUST implement 
// __SYSTEM.IQueryInterface. If IQueryInterface is not implemented,
// the type cannot be determined.
FUNCTION F_IsPointerToInterface : BOOL // TRUE if pointer appears to be an interface instance.
VAR_INPUT
	// Pointer to test.
	pValue : POINTER TO BYTE;
END_VAR
VAR
	pCheck : POINTER TO __UXINT;
END_VAR

pCheck := pValue;

CASE F_GetAddressMemoryArea(pCheck) OF 
	E_AddressMemoryArea.Static,
	E_AddressMemoryArea.Dynamic:
		pCheck := pCheck^;
ELSE
	RETURN;
	END_CASE
	
CASE F_GetAddressMemoryArea(pCheck) OF 
	E_AddressMemoryArea.Static,
	E_AddressMemoryArea.Dynamic:
		pCheck := pCheck^;
ELSE
	RETURN;
	END_CASE
	
CASE F_GetAddressMemoryArea(pCheck) OF 
	E_AddressMemoryArea.Static,
	E_AddressMemoryArea.Dynamic:
		F_IsPointerToInterface := pCheck^ = SIZEOF(__UXINT);
	END_CASE

END_FUNCTION

// ---- POUs/F_ExtractVariableNameFromPath.TcPOU
// Extracts the variable name from a given variable/symbol path.
// [example] 'MAIN.bVar' -> 'bVar'
FUNCTION F_ExtractVariableNameFromPath : STRING // The variable name.
VAR_INPUT CONSTANT
	Path : Tc2_System.T_MaxString; // Variable/Symbol path. 
END_VAR
VAR
	pCursor : POINTER TO BYTE;
	pName : POINTER TO STRING;
END_VAR

pCursor := ADR(Path);

REPEAT
	CASE pCursor^ OF
		9..11, 13: RETURN;
		46: pName := pCursor + 1;
		END_CASE
	pCursor := pCursor + 1;
UNTIL	
	pCursor^ = 0
	END_REPEAT
	
F_ExtractVariableNameFromPath := SEL(pName <> 0, '', pName^);

END_FUNCTION

// ---- POUs/F_GetCurrentTaskCycleTime.TcPOU
(*
Returns the cycle time of the task that calls this function.

The value is retrieved at runtime and reflects the actual configured cycle time
of the calling task. Returns ``LTIME#0`` if called outside of a task context.
*)
FUNCTION F_GetCurrentTaskCycleTime : LTIME
VAR
	fbGetCurrentTaskIndex : Tc2_System.GETCURTASKINDEX;
END_VAR

fbGetCurrentTaskIndex();
F_GetCurrentTaskCycleTime := TO_LTIME(
	TwinCAT_SystemInfoVarList._TaskInfo[fbGetCurrentTaskIndex.Index].CycleTime * 100);

END_FUNCTION

// ---- POUs/F_GetCurrentTaskIndex.TcPOU
(*
Returns the index of the task that calls this function.

..note:: Falls back to task index 1 if  called outside the real-time context.
*)
FUNCTION F_GetCurrentTaskIndex : DINT
VAR
	fbGetCurrentTaskIndex : Tc2_System.GETCURTASKINDEX;
END_VAR

fbGetCurrentTaskIndex();
F_GetCurrentTaskIndex := fbGetCurrentTaskIndex.Index;

END_FUNCTION

// ---- POUs/F_GetInf.TcPOU
// Retrieves the positive infinity value for LREAL data type.
FUNCTION F_GetInf : LREAL // The positive infinity value.
VAR_STAT
	fInf : LREAL := TO_LREAL('#Inf');
END_VAR

F_GetInf := fInf;

END_FUNCTION

// ---- POUs/F_GetMemorySegment.TcPOU
//	Retrieves the memory address of a segment of memory.
FUNCTION F_GetMemorySegment : POINTER TO BYTE // A pointer to the memory location of the specified segment.
VAR_INPUT
    pAddress : POINTER TO BYTE; // Starting address of the memory location.
    Size     : T_Size; // Size of one segment.
    Index    : T_Position; // Index of the segment.
END_VAR

F_GetMemorySegment := SEL(pAddress <> 0, 0, pAddress + (Size * F_PositionToSize(Index)));

END_FUNCTION

// ---- POUs/F_GetNaN.TcPOU
// Retrieves the "Not-a-Number" (NaN) value for LREAL data type.
FUNCTION F_GetNaN : LREAL // The NaN value.
VAR_STAT
	fNaN : LREAL := TO_LREAL('#NaN');
END_VAR

F_GetNaN := fNaN;

END_FUNCTION

// ---- POUs/F_DeallocateMemory.TcPOU
// Safely releases a memory pointer. 
// Ensuring that dynamically allocated memory is properly deallocated,
// and statically allocated memory pointers are safely nullified to avoid potential memory issues.
FUNCTION F_DeallocateMemory
VAR_IN_OUT
	pAddress : POINTER TO BYTE; // The memory pointer to be released.
END_VAR

IF NOT __ISVALIDREF(pAddress) THEN RETURN; END_IF

CASE Tc2_System.F_CheckMemoryArea(pAddress, 1) OF
	Tc2_System.E_TcMemoryArea.Dynamic:
		__DELETE(pAddress); 
ELSE
	pAddress := 0;
	END_CASE

END_FUNCTION

// ---- POUs/F_GetTypeID.TcPOU
// Retrieves the type identifier for any variable.
// [note]
// This relies on heuristics and may require the FB to implement 
// __SYSTEM.IQueryInterface for reliable detection.
FUNCTION F_GetTypeID : T_TypeID // The unique Type ID or TypeClass value.
VAR_INPUT
	// The variable to inspect.
	Variable : ANY;
END_VAR
VAR
END_VAR

F_GetTypeID := F_GetTypeIDFromGeneric(Variable);

END_FUNCTION

// ---- POUs/F_GetTypeIDFromGeneric.TcPOU
// Retrieves the type identifier for a generic variable.
// [note]
// This relies on heuristics and may require the FB to implement 
// __SYSTEM.IQueryInterface for reliable detection.
FUNCTION F_GetTypeIDFromGeneric : T_TypeID // The unique Type ID or TypeClass value.
VAR_INPUT
	// The generic variable descriptor to inspect.
	Variable : T_Generic;
END_VAR
VAR
	pFB 	 : POINTER TO __UXINT;
END_VAR

IF Variable.pValue = 0 THEN 
	F_GetTypeIDFromGeneric := T_TypeClass.TYPE_NONE; 
	RETURN; 
	END_IF

CASE Variable.TypeClass OF
	T_TypeClass.TYPE_USERDEF:
		IF F_IsPointerToInterface(Variable.pValue) THEN 
			F_GetTypeIDFromGeneric := 100;
		ELSIF F_IsPointerToFunctionBlock(Variable.pValue) THEN 
			pFB := Variable.pValue;
			F_GetTypeIDFromGeneric := pFB^;
		ELSE 
			F_GetTypeIDFromGeneric := T_TypeClass.TYPE_USERDEF; 
			END_IF
ELSE
	F_GetTypeIDFromGeneric := Variable.TypeClass;
	END_CASE

END_FUNCTION

// ---- POUs/F_IsPointerToFunctionBlock.TcPOU
// Tries to guess if the given pointer refers to a function block instance. 
// [note] 
// This is heuristic and can be inaccurate. The FB MUST implement 
// __SYSTEM.IQueryInterface. If the FB does not implement IQueryInterface,
// its type cannot be determined.
FUNCTION F_IsPointerToFunctionBlock : BOOL // TRUE if pointer appears to be a function block instance.
VAR_INPUT
	// Pointer to test.
	pValue : POINTER TO BYTE;
END_VAR
VAR
	pCheck : POINTER TO __UXINT;
END_VAR

pCheck := pValue;

CASE F_GetAddressMemoryArea(pCheck) OF 
	E_AddressMemoryArea.Static,
	E_AddressMemoryArea.Dynamic:
		pCheck := pCheck^;
ELSE
	RETURN;
	END_CASE
	
CASE F_GetAddressMemoryArea(pCheck) OF 
	E_AddressMemoryArea.Static,
	E_AddressMemoryArea.Dynamic:
		F_IsPointerToFunctionBlock := pCheck^ = SIZEOF(__UXINT);
	END_CASE

END_FUNCTION

// ---- POUs/F_GetVariablePathByAddress.TcPOU
// Retrieves path of a variable using its memory address and size.
// [note] Variables allocated in dynamic memory are not supported.
{warning disable C0394}
FUNCTION F_GetVariablePathByAddress : Tc2_System.T_MaxString // The path of the variable.
VAR_INPUT CONSTANT
	pAddress 	: POINTER TO BYTE; // Memory address pointer of variable.
	Size 		: T_Size; // Size of variable (in bytes).
END_VAR
VAR_STAT
	nTmp : UDINT := SIZEOF(F_GetVariablePathByAddress);
END_VAR
VAR
	ipInterface : ITcIecApplicationInfo;
END_VAR

CASE Tc2_System.F_CheckMemoryArea(pAddress, 1) OF
	Tc2_System.E_TcMemoryArea.Dynamic: F_GetVariablePathByAddress := '<dynamic>';
	Tc2_System.E_TcMemoryArea.Unknown: F_GetVariablePathByAddress := '<unknown>';
ELSE
	IF NOT F_TcComIecApplicationInfo().GetInterface(ipInterface) THEN RETURN; END_IF
	ipInterface.GetSymbolNameByAddress(
		Size, pAddress, nTmp, ADR(F_GetVariablePathByAddress));
	END_CASE

END_FUNCTION

// ---- POUs/F_GetVariablePath.TcPOU
// Retrieves path of the specified variable.
// [note] Variables allocated in dynamic memory are not supported.
{warning disable C0394}
FUNCTION F_GetVariablePath : Tc2_System.T_MaxString // The path of the variable.
VAR_INPUT
	 Variable : ANY; // The variable whose path is to be determined.
END_VAR
VAR_STAT
	nTmp : UDINT := SIZEOF(F_GetVariablePath);
END_VAR
VAR
	ipInterface : ITcIecApplicationInfo;
END_VAR

CASE Tc2_System.F_CheckMemoryArea(Variable.pValue, 1) OF
	Tc2_System.E_TcMemoryArea.Dynamic: F_GetVariablePath := '<dynamic>';
	Tc2_System.E_TcMemoryArea.Unknown: F_GetVariablePath := '<unknown>';
ELSE
	IF NOT F_TcComIecApplicationInfo().GetInterface(ipInterface) THEN RETURN; END_IF
	ipInterface.GetSymbolNameByAddress(
		TO_UDINT(Variable.diSize), Variable.pValue, nTmp, ADR(F_GetVariablePath));
	END_CASE

END_FUNCTION

// ---- POUs/F_AllAreTrue.TcPOU
// Checks if all elements in a boolean array are true.
FUNCTION F_AllAreTrue : BOOL // True if all elements in the array are true.
VAR_IN_OUT
	arValues : ARRAY[*] OF BOOL; // An array of boolean values to check.
END_VAR
VAR
	i : T_Position;
END_VAR

FOR i := LOWER_BOUND(arValues, 1) TO UPPER_BOUND(arValues, 1) DO
	IF NOT arValues[i] THEN RETURN; END_IF 
	END_FOR
	
F_AllAreTrue := TRUE;

END_FUNCTION

// ---- POUs/F_Lerp.TcPOU
// Linearly interpolates between two values based on a given percentage.
FUNCTION F_Lerp : LREAL // The interpolated value.
VAR_INPUT
    fStartValue : LREAL; // The starting value.
    fEndValue   : LREAL; // The ending value.
    fPercentage : LREAL; // The interpolation factor (0.0 to 1.0).
END_VAR

F_Lerp := fStartValue + (fEndValue - fStartValue) * fPercentage;

END_FUNCTION

// ---- POUs/F_RunAllRunnables.TcPOU
(*
Calls :meth:`I_Runnable.Run` on every non-null entry in the given array.

Entries set to ``0`` are skipped, so sparse arrays are safe to pass in.
The array bounds are read at runtime, so any fixed size array is accepted.
*)
FUNCTION F_RunAllRunnables
VAR_IN_OUT
	// Reference to the array containing the runnables to run.
	arRunnables : ARRAY[*] OF I_Runnable;
END_VAR
VAR
	i : T_Position;
END_VAR

FOR i := LOWER_BOUND(arRunnables, 1) TO UPPER_BOUND(arRunnables, 1) DO
	IF arRunnables[i] = 0 THEN CONTINUE; END_IF
	arRunnables[i].Run();
END_FOR

END_FUNCTION

// ---- POUs/F_SetOnFalse.TcPOU
// Sets the boolean value to true if it is false and returns true if it was false before being set.
FUNCTION F_SetOnFalse : BOOL // Whether the value was false before setting.
VAR_INPUT
    bValue : REFERENCE TO BOOL; // Boolean value to set.
END_VAR

F_SetOnFalse 	:= NOT bValue;
bValue 			:= TRUE;

END_FUNCTION

// ---- POUs/F_SwapMemory.TcPOU
// Swaps the contents of two memory locations.
FUNCTION F_SwapMemory
VAR_INPUT
    pAddress1 	: POINTER TO BYTE; // Pointer to the first memory location.
    pAddress2 	: POINTER TO BYTE; // Pointer to the second memory location.
    Size 		: T_Size;          // Size of each memory element (in bytes).
END_VAR
VAR
	i, End 			: T_Position;
	nTmp 			: __XWORD;
	pTmpAddress1	: POINTER TO __XWORD := pAddress1;	
	pTmpAddress2	: POINTER TO __XWORD := pAddress2;
END_VAR

IF pAddress1 = pAddress2 OR pAddress1 = 0 OR pAddress2 = 0 THEN RETURN; END_IF

End := TO_LINT(Size / SIZEOF(__XWORD)) - 1;
FOR i := 0 TO End DO
	nTmp := pTmpAddress1[i];
	pTmpAddress1[i] := pTmpAddress2[i];
	pTmpAddress2[i] := nTmp;
	END_FOR

End := TO_LINT(Size) - 1;
FOR i := i TO End DO
	nTmp := pAddress1[i];
	pAddress1[i] := pAddress2[i];
	pAddress2[i] := TO_BYTE(nTmp);
	END_FOR

END_FUNCTION

// ---- POUs/F_GetTypeNameByAddress.TcPOU
// Retrieves the datatype of a variable as a string using its pointer and size.
// [note] Variables allocated in dynamic memory are not supported.
{warning disable C0394}
FUNCTION F_GetTypeNameByAddress : STRING // The datatype name of the variable as a string.
VAR_INPUT CONSTANT
	pAddress 	: POINTER TO BYTE; // Memory address pointer of variable.
	Size 		: T_Size; // Size of variable (in bytes).
END_VAR
VAR_STAT
	nTmp : UDINT := SIZEOF(F_GetTypeNameByAddress);
END_VAR
VAR
	ipInterface : ITcIecApplicationInfo;
END_VAR

CASE Tc2_System.F_CheckMemoryArea(pAddress, 1) OF
	Tc2_System.E_TcMemoryArea.Dynamic: F_GetTypeNameByAddress := '<dynamic>';
	Tc2_System.E_TcMemoryArea.Unknown: F_GetTypeNameByAddress := '<unknown>';
ELSE
	IF NOT F_TcComIecApplicationInfo().GetInterface(ipInterface) THEN RETURN; END_IF
	ipInterface.GetDatatypeNameByAddress(
		Size, pAddress, nTmp, ADR(F_GetTypeNameByAddress));
	END_CASE

END_FUNCTION

// ---- POUs/F_GetTypeNameByPath.TcPOU
// Retrieves the datatype of a variable as a string given its path.
{warning disable C0394}
FUNCTION F_GetTypeNameByPath : STRING // The datatype name of the variable as a string.
VAR_INPUT
	// Variable/Symbol path as string.
	// [example] 'MAIN.bVar'.
	Path : Tc2_System.T_MaxString; 
END_VAR
VAR_STAT
	nTmp : UDINT := SIZEOF(F_GetTypeNameByPath);
END_VAR 
VAR
	ipInterface : ITcIecApplicationInfo;
END_VAR

IF NOT F_TcComIecApplicationInfo().GetInterface(ipInterface) THEN RETURN; END_IF

ipInterface.GetSymbolDatatype(Path, nTmp, ADR(F_GetTypeNameByPath));

END_FUNCTION

// ---- POUs/F_RoundToDecimalPlaces.TcPOU
// Rounds a given floating-point number to a specified number of decimal places.
FUNCTION F_RoundToDecimalPlaces : LREAL // The rounded floating-point value with the specified number of decimal places.
VAR_INPUT
	fValue 			: LREAL; // The floating-point value to be rounded.
	nDecimalPlaces 	: USINT; // The number of decimal places to round to.
END_VAR
VAR
	fMultiplier, 
	fTrunc 			: LREAL;
END_VAR

fMultiplier := EXPT(10, nDecimalPlaces);
F_RoundToDecimalPlaces := LIMIT(GVL_TypeValueLimits.LREAL_MIN, fValue * fMultiplier, GVL_TypeValueLimits.LREAL_MIN);
fTrunc := F_TruncateNumber(F_RoundToDecimalPlaces);

F_RoundToDecimalPlaces := 
	(fTrunc + SEL(F_RoundToDecimalPlaces - fTrunc >= 0.5, 0, 1)) / fMultiplier;

END_FUNCTION

// ---- POUs/F_TryDerefPointer.TcPOU
// Attempts to dereference a pointer up to a given number of levels.
// [note] the given pointer is returned if Levels is 0.
FUNCTION F_TryDerefPointer : POINTER TO BYTE // Final dereferenced readable pointer.
VAR_INPUT
	// Pointer to start dereferencing from.
	pValue : POINTER TO BYTE;
	// Number of dereference levels to attempt.
	Levels : T_Size;
END_VAR
VAR
	i 		: T_Position;
	pTmp 	: POINTER TO POINTER TO BYTE;
END_VAR

// Return the same pointer of 0 levels.
pTmp := F_TryDerefPointer := pValue;

FOR i := 1 TO Levels DO
	RETURN(NOT F_IsReadablePointer(F_TryDerefPointer));
	pTmp := F_TryDerefPointer;
	F_TryDerefPointer := pTmp^;
	END_FOR

END_FUNCTION

// ---- Project Information/F_GetCompany.TcPOU
// This function has been automatically generated from the project information.
{attribute 'signature_flag' := '1073741824'}
{attribute 'TcGenerated'}
{attribute 'no-analysis'}
FUNCTION F_GetCompany : WSTRING
VAR_INPUT
	
END_VAR

F_GetCompany := "FisoThemes";

END_FUNCTION

// ---- Project Information/F_GetTitle.TcPOU
// This function has been automatically generated from the project information.
{attribute 'signature_flag' := '1073741824'}
{attribute 'TcGenerated'}
{attribute 'no-analysis'}
FUNCTION F_GetTitle : WSTRING
VAR_INPUT
	
END_VAR

F_GetTitle := "FsCommon";

END_FUNCTION

// ---- Project Information/F_GetVersion.TcPOU
// This function has been automatically generated from the project information.
{attribute 'signature_flag' := '1073741824'}
{attribute 'TcGenerated'}
{attribute 'no-analysis'}
FUNCTION F_GetVersion : ST_LibVersion
VAR_INPUT
	
END_VAR

F_GetVersion.iMajor := 0;
F_GetVersion.iMinor := 7;
F_GetVersion.iBuild := 0;
F_GetVersion.iRevision := 0;
F_GetVersion.sVersion := '0.7.0';
F_GetVersion.nFlags := 0;

END_FUNCTION
